LIN {X 0,Y 305.463,Z 118.06,A -85,B 0,C 180,E1 -16139.051,E2 -16139.051} C_VEL
LIN {X 0,Y 305.415,Z 118.064,A -85,B 0,C 180,E1 -16141.953,E2 -16141.953} C_VEL
LIN {X 0,Y 305.449,Z 118.063,A -85,B 0,C 180,E1 -16145.112,E2 -16145.112} C_VEL
LIN {X 0,Y 305.493,Z 118.055,A -85,B 0,C 180,E1 -16146.531,E2 -16146.531} C_VEL
LIN {X 0,Y 304.825,Z 118.142,A -85,B 0,C 180,E1 -16147.631,E2 -16147.631} C_VEL
LIN {X 0,Y 301.946,Z 118.499,A -85,B 0,C 180,E1 -16149.419,E2 -16149.419} C_VEL
LIN {X 0,Y 299.512,Z 118.803,A -85,B 0,C 180,E1 -16150.871,E2 -16150.871} C_VEL
LIN {X 0,Y 298.486,Z 118.925,A -85,B 0,C 180,E1 -16151.996,E2 -16151.996} C_VEL
LIN {X 0,Y 298.412,Z 118.928,A -85,B 0,C 180,E1 -16152.377,E2 -16152.377} C_VEL
LIN {X 0,Y 298.464,Z 118.93,A -85,B 0,C 180,E1 -16155.064,E2 -16155.064} C_VEL
LIN {X 0,Y 298.429,Z 118.934,A -85,B 0,C 180,E1 -16158.9,E2 -16158.9} C_VEL
LIN {X 0,Y 298.444,Z 118.927,A -85,B 0,C 180,E1 -16163.189,E2 -16163.189} C_VEL
LIN {X 0,Y 298.373,Z 118.94,A -85,B 0,C 180,E1 -16167.204,E2 -16167.204} C_VEL
LIN {X 0,Y 298.409,Z 118.927,A -85,B 0,C 180,E1 -16170.618,E2 -16170.618} C_VEL
LIN {X 0,Y 298.463,Z 118.924,A -85,B 0,C 180,E1 -16173.477,E2 -16173.477} C_VEL
LIN {X 0,Y 298.499,Z 118.926,A -85,B 0,C 180,E1 -16176.664,E2 -16176.664} C_VEL
LIN {X 0,Y 298.548,Z 118.918,A -85,B 0,C 180,E1 -16180.763,E2 -16180.763} C_VEL
LIN {X 0,Y 298.576,Z 118.913,A -85,B 0,C 180,E1 -16184.999,E2 -16184.999} C_VEL
LIN {X 0,Y 298.58,Z 118.916,A -85,B 0,C 180,E1 -16189.151,E2 -16189.151} C_VEL
LIN {X 0,Y 298.744,Z 118.888,A -85,B 0,C 180,E1 -16191.89,E2 -16191.89} C_VEL
LIN {X 0,Y 298.65,Z 118.896,A -85,B 0,C 180,E1 -16194.603,E2 -16194.603} C_VEL
LIN {X 0,Y 298.917,Z 118.873,A -85,B 0,C 180,E1 -16198.657,E2 -16198.657} C_VEL
LIN {X 0,Y 298.915,Z 118.874,A -85,B 0,C 180,E1 -16201.352,E2 -16201.352} C_VEL
LIN {X 0,Y 298.789,Z 118.885,A -85,B 0,C 180,E1 -16206.758,E2 -16206.758} C_VEL
LIN {X 0,Y 298.673,Z 118.905,A -85,B 0,C 180,E1 -16209.485,E2 -16209.485} C_VEL
LIN {X 0,Y 298.546,Z 118.92,A -85,B 0,C 180,E1 -16213.62,E2 -16213.62} C_VEL
LIN {X 0,Y 298.544,Z 118.921,A -85,B 0,C 180,E1 -16216.413,E2 -16216.413} C_VEL
LIN {X 0,Y 298.508,Z 118.924,A -85,B 0,C 180,E1 -16219.659,E2 -16219.659} C_VEL
LIN {X 0,Y 298.455,Z 118.93,A -85,B 0,C 180,E1 -16223.602,E2 -16223.602} C_VEL
LIN {X 0,Y 298.488,Z 118.928,A -85,B 0,C 180,E1 -16226.578,E2 -16226.578} C_VEL
LIN {X 0,Y 298.42,Z 118.934,A -85,B 0,C 180,E1 -16229.645,E2 -16229.645} C_VEL
LIN {X 0,Y 298.395,Z 118.938,A -85,B 0,C 180,E1 -16232.804,E2 -16232.804} C_VEL
LIN {X 0,Y 298.447,Z 118.932,A -85,B 0,C 180,E1 -16236.811,E2 -16236.811} C_VEL
LIN {X 0,Y 298.41,Z 118.936,A -85,B 0,C 180,E1 -16239.49,E2 -16239.49} C_VEL
LIN {X 0,Y 298.401,Z 118.939,A -85,B 0,C 180,E1 -16243.107,E2 -16243.107} C_VEL
LIN {X 0,Y 298.406,Z 118.938,A -85,B 0,C 180,E1 -16246.924,E2 -16246.924} C_VEL
LIN {X 0,Y 298.408,Z 118.938,A -85,B 0,C 180,E1 -16251.01,E2 -16251.01} C_VEL
LIN {X 0,Y 298.469,Z 119.026,A -85,B 0,C 180,E1 -16254.32,E2 -16254.32} C_VEL
LIN {X 0,Y 301.25,Z 131.247,A -85,B 0,C 180,E1 -16257.947,E2 -16257.947} C_VEL
LIN {X 0,Y 302.367,Z 136.348,A -85,B 0,C 180,E1 -16259.403,E2 -16259.403} C_VEL
LIN {X 0,Y 308.581,Z 152.762,A -85,B 0,C 180,E1 -16260.374,E2 -16260.374} C_VEL
LIN {X 0,Y 313.309,Z 184.218,A -85,B 0,C 180,E1 -16261.555,E2 -16261.555} C_VEL
LIN {X 0,Y 310.762,Z 275.009,A -85,B 0,C 180,E1 -16263.654,E2 -16263.654} C_VEL
LIN {X 0,Y 309.864,Z 288.738,A -85,B 0,C 180,E1 -16264.205,E2 -16264.205} C_VEL
LIN {X 0,Y 308.586,Z 302.3,A -85,B 0,C 180,E1 -16264.993,E2 -16264.993} C_VEL
LIN {X 0,Y 307.177,Z 315.166,A -85,B 0,C 180,E1 -16266.002,E2 -16266.002} C_VEL
LIN {X 0,Y 305.517,Z 328.379,A -85,B 0,C 180,E1 -16267.339,E2 -16267.339} C_VEL
LIN {X 0,Y 303.999,Z 338.844,A -85,B 0,C 180,E1 -16268.649,E2 -16268.649} C_VEL
LIN {X 0,Y 302.26,Z 349.716,A -85,B 0,C 180,E1 -16270.299,E2 -16270.299} C_VEL
LIN {X 0,Y 300.609,Z 360.479,A -85,B 0,C 180,E1 -16272.308,E2 -16272.308} C_VEL
LIN {X 0,Y 299.312,Z 369.247,A -85,B 0,C 180,E1 -16274.311,E2 -16274.311} C_VEL
LIN {X 0,Y 298.447,Z 375.565,A -85,B 0,C 180,E1 -16276.034,E2 -16276.034} C_VEL
LIN {X 0,Y 297.482,Z 382.796,A -85,B 0,C 180,E1 -16278.418,E2 -16278.418} C_VEL
LIN {X 0,Y 296.859,Z 389.274,A -85,B 0,C 180,E1 -16281.15,E2 -16281.15} C_VEL
LIN {X 0,Y 296.62,Z 392.996,A -85,B 0,C 180,E1 -16283.198,E2 -16283.198} C_VEL
LIN {X 0,Y 296.508,Z 396.618,A -85,B 0,C 180,E1 -16285.924,E2 -16285.924} C_VEL
LIN {X 0,Y 296.53,Z 397.888,A -85,B 0,C 180,E1 -16287.285,E2 -16287.285} C_VEL
LIN {X 0,Y 296.524,Z 399.388,A -85,B 0,C 180,E1 -16290.002,E2 -16290.002} C_VEL
LIN {X 0,Y 296.525,Z 399.54,A -85,B 0,C 180,E1 -16292.719,E2 -16292.719} C_VEL
LIN {X 0,Y 296.525,Z 398.363,A -85,B 0,C 180,E1 -16295.442,E2 -16295.442} C_VEL
LIN {X 0,Y 296.863,Z 395.854,A -85,B 0,C 180,E1 -16298.168,E2 -16298.168} C_VEL
LIN {X 0,Y 297.526,Z 391.948,A -85,B 0,C 180,E1 -16300.895,E2 -16300.895} C_VEL
LIN {X 0,Y 298.381,Z 387.999,A -85,B 0,C 180,E1 -16302.932,E2 -16302.932} C_VEL
LIN {X 0,Y 299.567,Z 383.169,A -85,B 0,C 180,E1 -16304.957,E2 -16304.957} C_VEL
LIN {X 0,Y 301.265,Z 376.222,A -85,B 0,C 180,E1 -16307.312,E2 -16307.312} C_VEL
LIN {X 0,Y 303.49,Z 367.688,A -85,B 0,C 180,E1 -16309.622,E2 -16309.622} C_VEL
LIN {X 0,Y 305.826,Z 358.785,A -85,B 0,C 180,E1 -16311.575,E2 -16311.575} C_VEL
LIN {X 0,Y 308.109,Z 349.971,A -85,B 0,C 180,E1 -16313.173,E2 -16313.173} C_VEL
LIN {X 0,Y 310.534,Z 339.507,A -85,B 0,C 180,E1 -16314.754,E2 -16314.754} C_VEL
LIN {X 0,Y 312.969,Z 328.052,A -85,B 0,C 180,E1 -16316.162,E2 -16316.162} C_VEL
LIN {X 0,Y 315.302,Z 315.733,A -85,B 0,C 180,E1 -16317.371,E2 -16317.371} C_VEL
LIN {X 0,Y 317.224,Z 303.024,A -85,B 0,C 180,E1 -16318.357,E2 -16318.357} C_VEL
LIN {X 0,Y 319.163,Z 288.698,A -85,B 0,C 180,E1 -16319.158,E2 -16319.158} C_VEL
LIN {X 0,Y 320.329,Z 275.633,A -85,B 0,C 180,E1 -16319.673,E2 -16319.673} C_VEL
LIN {X 0,Y 321.397,Z 250.364,A -85,B 0,C 180,E1 -16320.292,E2 -16320.292} C_VEL
LIN {X 0,Y 323.754,Z 186.86,A -85,B 0,C 180,E1 -16321.729,E2 -16321.729} C_VEL
LIN {X 0,Y 320.712,Z 169.862,A -85,B 0,C 180,E1 -16322.611,E2 -16322.611} C_VEL
LIN {X 0,Y 314.466,Z 156.405,A -85,B 0,C 180,E1 -16323.882,E2 -16323.882} C_VEL
LIN {X 0,Y 307.49,Z 143.185,A -85,B 0,C 180,E1 -16325.342,E2 -16325.342} C_VEL
LIN {X 0,Y 304.773,Z 138.364,A -85,B 0,C 180,E1 -16325.93,E2 -16325.93} C_VEL
LIN {X 0,Y 303.138,Z 135.112,A -85,B 0,C 180,E1 -16326.337,E2 -16326.337} C_VEL
LIN {X 0,Y 300.715,Z 126.551,A -85,B 0,C 180,E1 -16329.53,E2 -16329.53} C_VEL
LIN {X 0,Y 298.433,Z 118.935,A -85,B 0,C 180,E1 -16332.701,E2 -16332.701} C_VEL
LIN {X 0,Y 298.391,Z 118.937,A -85,B 0,C 180,E1 -16336.914,E2 -16336.914} C_VEL
LIN {X 0,Y 298.412,Z 118.938,A -85,B 0,C 180,E1 -16341.007,E2 -16341.007} C_VEL
LIN {X 0,Y 298.421,Z 118.938,A -85,B 0,C 180,E1 -16343.926,E2 -16343.926} C_VEL
LIN {X 0,Y 298.408,Z 118.94,A -85,B 0,C 180,E1 -16347.197,E2 -16347.197} C_VEL
LIN {X 0,Y 298.418,Z 118.938,A -85,B 0,C 180,E1 -16350.623,E2 -16350.623} C_VEL
LIN {X 0,Y 298.456,Z 118.93,A -85,B 0,C 180,E1 -16354.917,E2 -16354.917} C_VEL
LIN {X 0,Y 298.451,Z 118.924,A -85,B 0,C 180,E1 -16359.311,E2 -16359.311} C_VEL
LIN {X 0,Y 298.549,Z 118.922,A -85,B 0,C 180,E1 -16362.176,E2 -16362.176} C_VEL
LIN {X 0,Y 298.607,Z 118.908,A -85,B 0,C 180,E1 -16364.991,E2 -16364.991} C_VEL
LIN {X 0,Y 298.595,Z 118.909,A -85,B 0,C 180,E1 -16369.143,E2 -16369.143} C_VEL
LIN {X 0,Y 298.709,Z 118.893,A -85,B 0,C 180,E1 -16371.88,E2 -16371.88} C_VEL
LIN {X 0,Y 298.645,Z 118.911,A -85,B 0,C 180,E1 -16374.594,E2 -16374.594} C_VEL
LIN {X 0,Y 298.926,Z 118.876,A -85,B 0,C 180,E1 -16378.648,E2 -16378.648} C_VEL
LIN {X 0,Y 298.926,Z 118.862,A -85,B 0,C 180,E1 -16381.343,E2 -16381.343} C_VEL
LIN {X 0,Y 298.645,Z 118.899,A -85,B 0,C 180,E1 -16385.397,E2 -16385.397} C_VEL
LIN {X 0,Y 298.717,Z 118.898,A -85,B 0,C 180,E1 -16388.11,E2 -16388.11} C_VEL
LIN {X 0,Y 298.553,Z 118.917,A -85,B 0,C 180,E1 -16392.227,E2 -16392.227} C_VEL
LIN {X 0,Y 298.607,Z 118.916,A -85,B 0,C 180,E1 -16395.204,E2 -16395.204} C_VEL
LIN {X 0,Y 298.538,Z 118.92,A -85,B 0,C 180,E1 -16399.238,E2 -16399.238} C_VEL
LIN {X 0,Y 298.454,Z 118.929,A -85,B 0,C 180,E1 -16403.592,E2 -16403.592} C_VEL
LIN {X 0,Y 298.48,Z 118.925,A -85,B 0,C 180,E1 -16406.569,E2 -16406.569} C_VEL
LIN {X 0,Y 298.397,Z 118.919,A -85,B 0,C 180,E1 -16409.637,E2 -16409.637} C_VEL
LIN {X 0,Y 298.384,Z 118.937,A -85,B 0,C 180,E1 -16412.795,E2 -16412.795} C_VEL
LIN {X 0,Y 298.434,Z 119.032,A -85,B 0,C 180,E1 -16415.333,E2 -16415.333} C_VEL
LIN {X 0,Y 299.696,Z 123.328,A -85,B 0,C 180,E1 -16417.147,E2 -16417.147} C_VEL
LIN {X 0,Y 302.219,Z 127.458,A -85,B 0,C 180,E1 -16417.718,E2 -16417.718} C_VEL
LIN {X 0,Y 310.622,Z 141.607,A -85,B 0,C 180,E1 -16419.523,E2 -16419.523} C_VEL
LIN {X 0,Y 318.57,Z 156.631,A -85,B 0,C 180,E1 -16421.139,E2 -16421.139} C_VEL
LIN {X 0,Y 324.357,Z 169.063,A -85,B 0,C 180,E1 -16422.282,E2 -16422.282} C_VEL
LIN {X 0,Y 320.9,Z 259.44,A -85,B 0,C 180,E1 -16424.357,E2 -16424.357} C_VEL
LIN {X 0,Y 319.7,Z 273.914,A -85,B 0,C 180,E1 -16424.926,E2 -16424.926} C_VEL
LIN {X 0,Y 318.002,Z 288.36,A -85,B 0,C 180,E1 -16425.767,E2 -16425.767} C_VEL
LIN {X 0,Y 316.179,Z 301.192,A -85,B 0,C 180,E1 -16426.786,E2 -16426.786} C_VEL
LIN {X 0,Y 313.949,Z 313.553,A -85,B 0,C 180,E1 -16428.025,E2 -16428.025} C_VEL
LIN {X 0,Y 311.417,Z 325.585,A -85,B 0,C 180,E1 -16429.536,E2 -16429.536} C_VEL
LIN {X 0,Y 308.855,Z 336.611,A -85,B 0,C 180,E1 -16431.26,E2 -16431.26} C_VEL
LIN {X 0,Y 306.169,Z 347.321,A -85,B 0,C 180,E1 -16433.355,E2 -16433.355} C_VEL
LIN {X 0,Y 303.827,Z 356.079,A -85,B 0,C 180,E1 -16435.476,E2 -16435.476} C_VEL
LIN {X 0,Y 301.81,Z 363.266,A -85,B 0,C 180,E1 -16437.615,E2 -16437.615} C_VEL
LIN {X 0,Y 300.013,Z 369.838,A -85,B 0,C 180,E1 -16440.071,E2 -16440.071} C_VEL
LIN {X 0,Y 298.577,Z 375.202,A -85,B 0,C 180,E1 -16442.676,E2 -16442.676} C_VEL
LIN {X 0,Y 297.69,Z 378.573,A -85,B 0,C 180,E1 -16444.85,E2 -16444.85} C_VEL
LIN {X 0,Y 296.918,Z 381.627,A -85,B 0,C 180,E1 -16447.744,E2 -16447.744} C_VEL
LIN {X 0,Y 296.434,Z 383.173,A -85,B 0,C 180,E1 -16450.613,E2 -16450.613} C_VEL
LIN {X 0,Y 296.355,Z 383.402,A -85,B 0,C 180,E1 -16452.042,E2 -16452.042} C_VEL
LIN {X 0,Y 296.27,Z 382.793,A -85,B 0,C 180,E1 -16454.872,E2 -16454.872} C_VEL
LIN {X 0,Y 296.35,Z 381.8,A -85,B 0,C 180,E1 -16456.461,E2 -16456.461} C_VEL
LIN {X 0,Y 296.511,Z 379.191,A -85,B 0,C 180,E1 -16459.068,E2 -16459.068} C_VEL
LIN {X 0,Y 297.015,Z 374.96,A -85,B 0,C 180,E1 -16461.836,E2 -16461.836} C_VEL
LIN {X 0,Y 297.663,Z 369.164,A -85,B 0,C 180,E1 -16464.579,E2 -16464.579} C_VEL
LIN {X 0,Y 298.585,Z 362.628,A -85,B 0,C 180,E1 -16466.962,E2 -16466.962} C_VEL
LIN {X 0,Y 299.812,Z 354.531,A -85,B 0,C 180,E1 -16469.327,E2 -16469.327} C_VEL
LIN {X 0,Y 301.206,Z 346.043,A -85,B 0,C 180,E1 -16471.335,E2 -16471.335} C_VEL
LIN {X 0,Y 302.605,Z 337.211,A -85,B 0,C 180,E1 -16473.071,E2 -16473.071} C_VEL
LIN {X 0,Y 304.139,Z 326.644,A -85,B 0,C 180,E1 -16474.803,E2 -16474.803} C_VEL
LIN {X 0,Y 305.924,Z 314.369,A -85,B 0,C 180,E1 -16476.428,E2 -16476.428} C_VEL
LIN {X 0,Y 307.463,Z 302.214,A -85,B 0,C 180,E1 -16477.716,E2 -16477.716} C_VEL
LIN {X 0,Y 308.856,Z 288.771,A -85,B 0,C 180,E1 -16478.833,E2 -16478.833} C_VEL
LIN {X 0,Y 309.997,Z 274.732,A -85,B 0,C 180,E1 -16479.705,E2 -16479.705} C_VEL
LIN {X 0,Y 310.751,Z 261.089,A -85,B 0,C 180,E1 -16480.298,E2 -16480.298} C_VEL
LIN {X 0,Y 311.486,Z 239.443,A -85,B 0,C 180,E1 -16480.849,E2 -16480.849} C_VEL
LIN {X 0,Y 313.804,Z 159.13,A -85,B 0,C 180,E1 -16482.665,E2 -16482.665} C_VEL
LIN {X 0,Y 305.648,Z 137.375,A -85,B 0,C 180,E1 -16483.911,E2 -16483.911} C_VEL
LIN {X 0,Y 299.264,Z 122.065,A -85,B 0,C 180,E1 -16484.898,E2 -16484.898} C_VEL
LIN {X 0,Y 298.54,Z 118.93,A -85,B 0,C 180,E1 -16485.92,E2 -16485.92} C_VEL
LIN {X 0,Y 298.531,Z 118.927,A -85,B 0,C 180,E1 -16489.684,E2 -16489.684} C_VEL
LIN {X 0,Y 298.455,Z 118.935,A -85,B 0,C 180,E1 -16493.596,E2 -16493.596} C_VEL
LIN {X 0,Y 298.456,Z 118.931,A -85,B 0,C 180,E1 -16496.575,E2 -16496.575} C_VEL
LIN {X 0,Y 298.389,Z 118.941,A -85,B 0,C 180,E1 -16499.642,E2 -16499.642} C_VEL
LIN {X 0,Y 298.366,Z 118.944,A -85,B 0,C 180,E1 -16502.801,E2 -16502.801} C_VEL
LIN {X 0,Y 298.46,Z 118.933,A -85,B 0,C 180,E1 -16506.821,E2 -16506.821} C_VEL
LIN {X 0,Y 298.437,Z 118.934,A -85,B 0,C 180,E1 -16509.479,E2 -16509.479} C_VEL
LIN {X 0,Y 298.412,Z 118.928,A -85,B 0,C 180,E1 -16512.377,E2 -16512.377} C_VEL
LIN {X 0,Y 297.765,Z 119.011,A -85,B 0,C 180,E1 -16513.504,E2 -16513.504} C_VEL
LIN {X 0,Y 294.898,Z 119.372,A -85,B 0,C 180,E1 -16515.339,E2 -16515.339} C_VEL
LIN {X 0,Y 292.464,Z 119.68,A -85,B 0,C 180,E1 -16516.828,E2 -16516.828} C_VEL
LIN {X 0,Y 291.436,Z 119.805,A -85,B 0,C 180,E1 -16517.982,E2 -16517.982} C_VEL
LIN {X 0,Y 291.363,Z 119.816,A -85,B 0,C 180,E1 -16518.373,E2 -16518.373} C_VEL
LIN {X 0,Y 291.36,Z 119.804,A -85,B 0,C 180,E1 -16521.167,E2 -16521.167} C_VEL
LIN {X 0,Y 291.36,Z 119.816,A -85,B 0,C 180,E1 -16524.633,E2 -16524.633} C_VEL
LIN {X 0,Y 291.351,Z 119.816,A -85,B 0,C 180,E1 -16527.955,E2 -16527.955} C_VEL
LIN {X 0,Y 291.359,Z 119.801,A -85,B 0,C 180,E1 -16531.162,E2 -16531.162} C_VEL
LIN {X 0,Y 291.403,Z 119.809,A -85,B 0,C 180,E1 -16534.277,E2 -16534.277} C_VEL
LIN {X 0,Y 291.427,Z 119.807,A -85,B 0,C 180,E1 -16537.309,E2 -16537.309} C_VEL
LIN {X 0,Y 291.495,Z 119.799,A -85,B 0,C 180,E1 -16540.278,E2 -16540.278} C_VEL
LIN {X 0,Y 291.538,Z 119.79,A -85,B 0,C 180,E1 -16544.628,E2 -16544.628} C_VEL
LIN {X 0,Y 291.523,Z 119.794,A -85,B 0,C 180,E1 -16548.885,E2 -16548.885} C_VEL
LIN {X 0,Y 291.694,Z 119.767,A -85,B 0,C 180,E1 -16551.693,E2 -16551.693} C_VEL
LIN {X 0,Y 291.62,Z 119.77,A -85,B 0,C 180,E1 -16554.473,E2 -16554.473} C_VEL
LIN {X 0,Y 291.883,Z 119.749,A -85,B 0,C 180,E1 -16558.625,E2 -16558.625} C_VEL
LIN {X 0,Y 291.881,Z 119.749,A -85,B 0,C 180,E1 -16561.384,E2 -16561.384} C_VEL
LIN {X 0,Y 291.738,Z 119.763,A -85,B 0,C 180,E1 -16566.922,E2 -16566.922} C_VEL
LIN {X 0,Y 291.622,Z 119.782,A -85,B 0,C 180,E1 -16569.716,E2 -16569.716} C_VEL
LIN {X 0,Y 291.516,Z 119.795,A -85,B 0,C 180,E1 -16573.955,E2 -16573.955} C_VEL
LIN {X 0,Y 291.482,Z 119.801,A -85,B 0,C 180,E1 -16576.822,E2 -16576.822} C_VEL
LIN {X 0,Y 291.447,Z 119.804,A -85,B 0,C 180,E1 -16579.879,E2 -16579.879} C_VEL
LIN {X 0,Y 291.398,Z 119.811,A -85,B 0,C 180,E1 -16584.21,E2 -16584.21} C_VEL
LIN {X 0,Y 291.421,Z 119.803,A -85,B 0,C 180,E1 -16587.276,E2 -16587.276} C_VEL
LIN {X 0,Y 291.336,Z 119.82,A -85,B 0,C 180,E1 -16590.441,E2 -16590.441} C_VEL
LIN {X 0,Y 291.345,Z 119.816,A -85,B 0,C 180,E1 -16593.702,E2 -16593.702} C_VEL
LIN {X 0,Y 291.382,Z 119.812,A -85,B 0,C 180,E1 -16597.259,E2 -16597.259} C_VEL
LIN {X 0,Y 291.335,Z 119.815,A -85,B 0,C 180,E1 -16600.646,E2 -16600.646} C_VEL
LIN {X 0,Y 291.293,Z 119.826,A -85,B 0,C 180,E1 -16604.406,E2 -16604.406} C_VEL
LIN {X 0,Y 291.33,Z 119.816,A -85,B 0,C 180,E1 -16608.408,E2 -16608.408} C_VEL
LIN {X 0,Y 291.357,Z 119.817,A -85,B 0,C 180,E1 -16611.162,E2 -16611.162} C_VEL
LIN {X 0,Y 291.448,Z 119.827,A -85,B 0,C 180,E1 -16613.789,E2 -16613.789} C_VEL
LIN {X 0,Y 294.169,Z 131.986,A -85,B 0,C 180,E1 -16617.5,E2 -16617.5} C_VEL
LIN {X 0,Y 295.189,Z 136.326,A -85,B 0,C 180,E1 -16618.733,E2 -16618.733} C_VEL
LIN {X 0,Y 302.347,Z 155.276,A -85,B 0,C 180,E1 -16619.897,E2 -16619.897} C_VEL
LIN {X 0,Y 306.734,Z 184.058,A -85,B 0,C 180,E1 -16621.017,E2 -16621.017} C_VEL
LIN {X 0,Y 304.219,Z 273.974,A -85,B 0,C 180,E1 -16623.135,E2 -16623.135} C_VEL
LIN {X 0,Y 303.301,Z 287.998,A -85,B 0,C 180,E1 -16623.697,E2 -16623.697} C_VEL
LIN {X 0,Y 301.99,Z 301.707,A -85,B 0,C 180,E1 -16624.501,E2 -16624.501} C_VEL
LIN {X 0,Y 300.413,Z 315.56,A -85,B 0,C 180,E1 -16625.611,E2 -16625.611} C_VEL
LIN {X 0,Y 298.703,Z 328.667,A -85,B 0,C 180,E1 -16626.976,E2 -16626.976} C_VEL
LIN {X 0,Y 297.141,Z 339.053,A -85,B 0,C 180,E1 -16628.314,E2 -16628.314} C_VEL
LIN {X 0,Y 295.503,Z 348.87,A -85,B 0,C 180,E1 -16629.829,E2 -16629.829} C_VEL
LIN {X 0,Y 293.758,Z 359.745,A -85,B 0,C 180,E1 -16631.882,E2 -16631.882} C_VEL
LIN {X 0,Y 292.283,Z 369.374,A -85,B 0,C 180,E1 -16634.123,E2 -16634.123} C_VEL
LIN {X 0,Y 291.309,Z 376.142,A -85,B 0,C 180,E1 -16636.041,E2 -16636.041} C_VEL
LIN {X 0,Y 290.474,Z 382.31,A -85,B 0,C 180,E1 -16638.134,E2 -16638.134} C_VEL
LIN {X 0,Y 289.808,Z 388.851,A -85,B 0,C 180,E1 -16640.933,E2 -16640.933} C_VEL
LIN {X 0,Y 289.553,Z 392.631,A -85,B 0,C 180,E1 -16643.031,E2 -16643.031} C_VEL
LIN {X 0,Y 289.41,Z 396.306,A -85,B 0,C 180,E1 -16645.824,E2 -16645.824} C_VEL
LIN {X 0,Y 289.457,Z 397.603,A -85,B 0,C 180,E1 -16647.219,E2 -16647.219} C_VEL
LIN {X 0,Y 289.442,Z 399.155,A -85,B 0,C 180,E1 -16650.002,E2 -16650.002} C_VEL
LIN {X 0,Y 289.429,Z 399.356,A -85,B 0,C 180,E1 -16652.786,E2 -16652.786} C_VEL
LIN {X 0,Y 289.449,Z 398.229,A -85,B 0,C 180,E1 -16655.575,E2 -16655.575} C_VEL
LIN {X 0,Y 289.794,Z 395.774,A -85,B 0,C 180,E1 -16658.369,E2 -16658.369} C_VEL
LIN {X 0,Y 290.522,Z 391.935,A -85,B 0,C 180,E1 -16661.161,E2 -16661.161} C_VEL
LIN {X 0,Y 291.445,Z 388.04,A -85,B 0,C 180,E1 -16663.245,E2 -16663.245} C_VEL
LIN {X 0,Y 293.16,Z 381.467,A -85,B 0,C 180,E1 -16666.005,E2 -16666.005} C_VEL
LIN {X 0,Y 295.047,Z 374.192,A -85,B 0,C 180,E1 -16668.4,E2 -16668.4} C_VEL
LIN {X 0,Y 297.568,Z 365.215,A -85,B 0,C 180,E1 -16670.751,E2 -16670.751} C_VEL
LIN {X 0,Y 300.112,Z 355.84,A -85,B 0,C 180,E1 -16672.732,E2 -16672.732} C_VEL
LIN {X 0,Y 302.79,Z 345.5,A -85,B 0,C 180,E1 -16674.515,E2 -16674.515} C_VEL
LIN {X 0,Y 305.429,Z 334.274,A -85,B 0,C 180,E1 -16676.092,E2 -16676.092} C_VEL
LIN {X 0,Y 308.125,Z 321.608,A -85,B 0,C 180,E1 -16677.51,E2 -16677.51} C_VEL
LIN {X 0,Y 310.295,Z 309.477,A -85,B 0,C 180,E1 -16678.587,E2 -16678.587} C_VEL
LIN {X 0,Y 312.129,Z 297.413,A -85,B 0,C 180,E1 -16679.417,E2 -16679.417} C_VEL
LIN {X 0,Y 313.88,Z 282.469,A -85,B 0,C 180,E1 -16680.16,E2 -16680.16} C_VEL
LIN {X 0,Y 314.965,Z 268.57,A -85,B 0,C 180,E1 -16680.601,E2 -16680.601} C_VEL
LIN {X 0,Y 318.039,Z 188.05,A -85,B 0,C 180,E1 -16682.464,E2 -16682.464} C_VEL
LIN {X 0,Y 315.295,Z 172.701,A -85,B 0,C 180,E1 -16683.287,E2 -16683.287} C_VEL
LIN {X 0,Y 308.733,Z 158.563,A -85,B 0,C 180,E1 -16684.681,E2 -16684.681} C_VEL
LIN {X 0,Y 300.876,Z 143.736,A -85,B 0,C 180,E1 -16686.413,E2 -16686.413} C_VEL
LIN {X 0,Y 297.687,Z 138.447,A -85,B 0,C 180,E1 -16687.137,E2 -16687.137} C_VEL
LIN {X 0,Y 295.821,Z 134.869,A -85,B 0,C 180,E1 -16687.608,E2 -16687.608} C_VEL
LIN {X 0,Y 293.561,Z 127.111,A -85,B 0,C 180,E1 -16690.661,E2 -16690.661} C_VEL
LIN {X 0,Y 291.324,Z 119.821,A -85,B 0,C 180,E1 -16693.799,E2 -16693.799} C_VEL
LIN {X 0,Y 291.314,Z 119.807,A -85,B 0,C 180,E1 -16697.502,E2 -16697.502} C_VEL
LIN {X 0,Y 291.36,Z 119.817,A -85,B 0,C 180,E1 -16701.155,E2 -16701.155} C_VEL
LIN {X 0,Y 291.371,Z 119.816,A -85,B 0,C 180,E1 -16704.623,E2 -16704.623} C_VEL
LIN {X 0,Y 291.381,Z 119.812,A -85,B 0,C 180,E1 -16707.948,E2 -16707.948} C_VEL
LIN {X 0,Y 291.36,Z 119.815,A -85,B 0,C 180,E1 -16711.152,E2 -16711.152} C_VEL
LIN {X 0,Y 291.375,Z 119.815,A -85,B 0,C 180,E1 -16714.264,E2 -16714.264} C_VEL
LIN {X 0,Y 291.387,Z 119.811,A -85,B 0,C 180,E1 -16717.296,E2 -16717.296} C_VEL
LIN {X 0,Y 291.473,Z 119.792,A -85,B 0,C 180,E1 -16720.267,E2 -16720.267} C_VEL
LIN {X 0,Y 291.554,Z 119.783,A -85,B 0,C 180,E1 -16724.631,E2 -16724.631} C_VEL
LIN {X 0,Y 291.541,Z 119.785,A -85,B 0,C 180,E1 -16728.877,E2 -16728.877} C_VEL
LIN {X 0,Y 291.663,Z 119.772,A -85,B 0,C 180,E1 -16731.683,E2 -16731.683} C_VEL
LIN {X 0,Y 291.614,Z 119.786,A -85,B 0,C 180,E1 -16734.464,E2 -16734.464} C_VEL
LIN {X 0,Y 291.892,Z 119.751,A -85,B 0,C 180,E1 -16738.616,E2 -16738.616} C_VEL
LIN {X 0,Y 291.893,Z 119.738,A -85,B 0,C 180,E1 -16741.375,E2 -16741.375} C_VEL
LIN {X 0,Y 291.664,Z 119.774,A -85,B 0,C 180,E1 -16746.551,E2 -16746.551} C_VEL
LIN {X 0,Y 291.572,Z 119.781,A -85,B 0,C 180,E1 -16749.709,E2 -16749.709} C_VEL
LIN {X 0,Y 291.524,Z 119.79,A -85,B 0,C 180,E1 -16753.945,E2 -16753.945} C_VEL
LIN {X 0,Y 291.488,Z 119.793,A -85,B 0,C 180,E1 -16756.812,E2 -16756.812} C_VEL
LIN {X 0,Y 291.45,Z 119.798,A -85,B 0,C 180,E1 -16759.869,E2 -16759.869} C_VEL
LIN {X 0,Y 291.395,Z 119.812,A -85,B 0,C 180,E1 -16764.2,E2 -16764.2} C_VEL
LIN {X 0,Y 291.41,Z 119.812,A -85,B 0,C 180,E1 -16767.267,E2 -16767.267} C_VEL
LIN {X 0,Y 291.316,Z 119.802,A -85,B 0,C 180,E1 -16770.433,E2 -16770.433} C_VEL
LIN {X 0,Y 291.371,Z 119.987,A -85,B 0,C 180,E1 -16774.229,E2 -16774.229} C_VEL
LIN {X 0,Y 292.495,Z 123.617,A -85,B 0,C 180,E1 -16775.844,E2 -16775.844} C_VEL
LIN {X 0,Y 294.842,Z 127.48,A -85,B 0,C 180,E1 -16776.411,E2 -16776.411} C_VEL
LIN {X 0,Y 301.819,Z 138.719,A -85,B 0,C 180,E1 -16778.01,E2 -16778.01} C_VEL
LIN {X 0,Y 308.948,Z 151.389,A -85,B 0,C 180,E1 -16779.557,E2 -16779.557} C_VEL
LIN {X 0,Y 316.269,Z 166.096,A -85,B 0,C 180,E1 -16781.084,E2 -16781.084} C_VEL
LIN {X 0,Y 318.672,Z 171.401,A -85,B 0,C 180,E1 -16781.574,E2 -16781.574} C_VEL
LIN {X 0,Y 315.078,Z 259.814,A -85,B 0,C 180,E1 -16783.628,E2 -16783.628} C_VEL
LIN {X 0,Y 313.818,Z 274.5,A -85,B 0,C 180,E1 -16784.22,E2 -16784.22} C_VEL
LIN {X 0,Y 312.097,Z 288.475,A -85,B 0,C 180,E1 -16785.045,E2 -16785.045} C_VEL
LIN {X 0,Y 310.256,Z 300.988,A -85,B 0,C 180,E1 -16786.049,E2 -16786.049} C_VEL
LIN {X 0,Y 308.037,Z 312.92,A -85,B 0,C 180,E1 -16787.251,E2 -16787.251} C_VEL
LIN {X 0,Y 305.368,Z 325.134,A -85,B 0,C 180,E1 -16788.789,E2 -16788.789} C_VEL
LIN {X 0,Y 302.703,Z 336.224,A -85,B 0,C 180,E1 -16790.535,E2 -16790.535} C_VEL
LIN {X 0,Y 300.067,Z 346.259,A -85,B 0,C 180,E1 -16792.484,E2 -16792.484} C_VEL
LIN {X 0,Y 297.552,Z 355.242,A -85,B 0,C 180,E1 -16794.64,E2 -16794.64} C_VEL
LIN {X 0,Y 295.406,Z 362.623,A -85,B 0,C 180,E1 -16796.823,E2 -16796.823} C_VEL
LIN {X 0,Y 293.651,Z 368.666,A -85,B 0,C 180,E1 -16799.03,E2 -16799.03} C_VEL
LIN {X 0,Y 292.218,Z 373.509,A -85,B 0,C 180,E1 -16801.246,E2 -16801.246} C_VEL
LIN {X 0,Y 291.233,Z 376.946,A -85,B 0,C 180,E1 -16803.223,E2 -16803.223} C_VEL
LIN {X 0,Y 290.311,Z 380.195,A -85,B 0,C 180,E1 -16805.696,E2 -16805.696} C_VEL
LIN {X 0,Y 289.939,Z 381.596,A -85,B 0,C 180,E1 -16807.178,E2 -16807.178} C_VEL
LIN {X 0,Y 289.401,Z 383.276,A -85,B 0,C 180,E1 -16810.122,E2 -16810.122} C_VEL
LIN {X 0,Y 289.294,Z 383.57,A -85,B 0,C 180,E1 -16811.588,E2 -16811.588} C_VEL
LIN {X 0,Y 289.171,Z 383.095,A -85,B 0,C 180,E1 -16814.492,E2 -16814.492} C_VEL
LIN {X 0,Y 289.289,Z 381.216,A -85,B 0,C 180,E1 -16817.369,E2 -16817.369} C_VEL
LIN {X 0,Y 289.599,Z 377.895,A -85,B 0,C 180,E1 -16820.217,E2 -16820.217} C_VEL
LIN {X 0,Y 289.999,Z 374.4,A -85,B 0,C 180,E1 -16822.338,E2 -16822.338} C_VEL
LIN {X 0,Y 290.539,Z 370.008,A -85,B 0,C 180,E1 -16824.446,E2 -16824.446} C_VEL
LIN {X 0,Y 291.422,Z 363.633,A -85,B 0,C 180,E1 -16826.888,E2 -16826.888} C_VEL
LIN {X 0,Y 292.683,Z 355.705,A -85,B 0,C 180,E1 -16829.31,E2 -16829.31} C_VEL
LIN {X 0,Y 294.084,Z 347.414,A -85,B 0,C 180,E1 -16831.367,E2 -16831.367} C_VEL
LIN {X 0,Y 295.785,Z 337.062,A -85,B 0,C 180,E1 -16833.476,E2 -16833.476} C_VEL
LIN {X 0,Y 297.388,Z 326.376,A -85,B 0,C 180,E1 -16835.252,E2 -16835.252} C_VEL
LIN {X 0,Y 299.066,Z 315.332,A -85,B 0,C 180,E1 -16836.746,E2 -16836.746} C_VEL
LIN {X 0,Y 300.639,Z 303.382,A -85,B 0,C 180,E1 -16838.061,E2 -16838.061} C_VEL
LIN {X 0,Y 302.06,Z 290.237,A -85,B 0,C 180,E1 -16839.203,E2 -16839.203} C_VEL
LIN {X 0,Y 303.25,Z 276.628,A -85,B 0,C 180,E1 -16840.092,E2 -16840.092} C_VEL
LIN {X 0,Y 304.11,Z 262.667,A -85,B 0,C 180,E1 -16840.736,E2 -16840.736} C_VEL
LIN {X 0,Y 304.795,Z 243.568,A -85,B 0,C 180,E1 -16841.259,E2 -16841.259} C_VEL
LIN {X 0,Y 307.278,Z 160.711,A -85,B 0,C 180,E1 -16843.169,E2 -16843.169} C_VEL
LIN {X 0,Y 299.691,Z 140.407,A -85,B 0,C 180,E1 -16844.37,E2 -16844.37} C_VEL
LIN {X 0,Y 292.982,Z 124.529,A -85,B 0,C 180,E1 -16845.431,E2 -16845.431} C_VEL
LIN {X 0,Y 292.079,Z 122.181,A -85,B 0,C 180,E1 -16845.608,E2 -16845.608} C_VEL
LIN {X 0,Y 291.482,Z 119.807,A -85,B 0,C 180,E1 -16846.459,E2 -16846.459} C_VEL
LIN {X 0,Y 291.462,Z 119.806,A -85,B 0,C 180,E1 -16849.899,E2 -16849.899} C_VEL
LIN {X 0,Y 291.404,Z 119.81,A -85,B 0,C 180,E1 -16854.203,E2 -16854.203} C_VEL
LIN {X 0,Y 291.389,Z 119.811,A -85,B 0,C 180,E1 -16857.272,E2 -16857.272} C_VEL
LIN {X 0,Y 291.306,Z 119.821,A -85,B 0,C 180,E1 -16860.438,E2 -16860.438} C_VEL
LIN {X 0,Y 291.319,Z 119.821,A -85,B 0,C 180,E1 -16863.699,E2 -16863.699} C_VEL
LIN {X 0,Y 291.425,Z 119.809,A -85,B 0,C 180,E1 -16867.277,E2 -16867.277} C_VEL
LIN {X 0,Y 291.393,Z 119.813,A -85,B 0,C 180,E1 -16870.629,E2 -16870.629} C_VEL
LIN {X 0,Y 291.383,Z 119.804,A -85,B 0,C 180,E1 -16874.381,E2 -16874.381} C_VEL
LIN {X 0,Y 291.363,Z 119.816,A -85,B 0,C 180,E1 -16878.373,E2 -16878.373} C_VEL
LIN {X 0,Y 290.714,Z 119.901,A -85,B 0,C 180,E1 -16879.528,E2 -16879.528} C_VEL
LIN {X 0,Y 287.844,Z 120.252,A -85,B 0,C 180,E1 -16881.407,E2 -16881.407} C_VEL
LIN {X 0,Y 285.414,Z 120.55,A -85,B 0,C 180,E1 -16882.933,E2 -16882.933} C_VEL
LIN {X 0,Y 284.398,Z 120.678,A -85,B 0,C 180,E1 -16884.116,E2 -16884.116} C_VEL
LIN {X 0,Y 284.33,Z 120.689,A -85,B 0,C 180,E1 -16884.517,E2 -16884.517} C_VEL
LIN {X 0,Y 284.274,Z 120.693,A -85,B 0,C 180,E1 -16888.73,E2 -16888.73} C_VEL
LIN {X 0,Y 284.375,Z 120.678,A -85,B 0,C 180,E1 -16892.83,E2 -16892.83} C_VEL
LIN {X 0,Y 284.382,Z 120.685,A -85,B 0,C 180,E1 -16896.714,E2 -16896.714} C_VEL
LIN {X 0,Y 284.417,Z 120.68,A -85,B 0,C 180,E1 -16899.875,E2 -16899.875} C_VEL
LIN {X 0,Y 284.475,Z 120.67,A -85,B 0,C 180,E1 -16904.463,E2 -16904.463} C_VEL
LIN {X 0,Y 284.475,Z 120.672,A -85,B 0,C 180,E1 -16908.606,E2 -16908.606} C_VEL
LIN {X 0,Y 284.645,Z 120.646,A -85,B 0,C 180,E1 -16911.486,E2 -16911.486} C_VEL
LIN {X 0,Y 284.591,Z 120.645,A -85,B 0,C 180,E1 -16914.336,E2 -16914.336} C_VEL
LIN {X 0,Y 284.849,Z 120.625,A -85,B 0,C 180,E1 -16918.591,E2 -16918.591} C_VEL
LIN {X 0,Y 284.847,Z 120.624,A -85,B 0,C 180,E1 -16921.418,E2 -16921.418} C_VEL
LIN {X 0,Y 284.69,Z 120.642,A -85,B 0,C 180,E1 -16927.095,E2 -16927.095} C_VEL
LIN {X 0,Y 284.559,Z 120.662,A -85,B 0,C 180,E1 -16929.96,E2 -16929.96} C_VEL
LIN {X 0,Y 284.476,Z 120.673,A -85,B 0,C 180,E1 -16934.307,E2 -16934.307} C_VEL
LIN {X 0,Y 284.421,Z 120.679,A -85,B 0,C 180,E1 -16937.253,E2 -16937.253} C_VEL
LIN {X 0,Y 284.375,Z 120.686,A -85,B 0,C 180,E1 -16940.247,E2 -16940.247} C_VEL
LIN {X 0,Y 284.367,Z 120.685,A -85,B 0,C 180,E1 -16943.88,E2 -16943.88} C_VEL
LIN {X 0,Y 284.396,Z 120.678,A -85,B 0,C 180,E1 -16947.178,E2 -16947.178} C_VEL
LIN {X 0,Y 284.295,Z 120.692,A -85,B 0,C 180,E1 -16951.279,E2 -16951.279} C_VEL
LIN {X 0,Y 284.342,Z 120.688,A -85,B 0,C 180,E1 -16955.352,E2 -16955.352} C_VEL
LIN {X 0,Y 284.32,Z 120.695,A -85,B 0,C 180,E1 -16958.172,E2 -16958.172} C_VEL
LIN {X 0,Y 284.272,Z 120.7,A -85,B 0,C 180,E1 -16962.128,E2 -16962.128} C_VEL
LIN {X 0,Y 284.259,Z 120.703,A -85,B 0,C 180,E1 -16966.193,E2 -16966.193} C_VEL
LIN {X 0,Y 284.311,Z 120.698,A -85,B 0,C 180,E1 -16970.028,E2 -16970.028} C_VEL
LIN {X 0,Y 284.41,Z 120.848,A -85,B 0,C 180,E1 -16973.298,E2 -16973.298} C_VEL
LIN {X 0,Y 287.144,Z 132.928,A -85,B 0,C 180,E1 -16977.095,E2 -16977.095} C_VEL
LIN {X 0,Y 287.809,Z 135.936,A -85,B 0,C 180,E1 -16978.006,E2 -16978.006} C_VEL
LIN {X 0,Y 296.067,Z 157.207,A -85,B 0,C 180,E1 -16979.378,E2 -16979.378} C_VEL
LIN {X 0,Y 300.269,Z 185.672,A -85,B 0,C 180,E1 -16980.509,E2 -16980.509} C_VEL
LIN {X 0,Y 297.637,Z 274.127,A -85,B 0,C 180,E1 -16982.634,E2 -16982.634} C_VEL
LIN {X 0,Y 296.706,Z 288.028,A -85,B 0,C 180,E1 -16983.208,E2 -16983.208} C_VEL
LIN {X 0,Y 295.284,Z 302.247,A -85,B 0,C 180,E1 -16984.068,E2 -16984.068} C_VEL
LIN {X 0,Y 293.734,Z 315.075,A -85,B 0,C 180,E1 -16985.117,E2 -16985.117} C_VEL
LIN {X 0,Y 292.1,Z 327.49,A -85,B 0,C 180,E1 -16986.424,E2 -16986.424} C_VEL
LIN {X 0,Y 290.483,Z 338.05,A -85,B 0,C 180,E1 -16987.79,E2 -16987.79} C_VEL
LIN {X 0,Y 288.783,Z 348.005,A -85,B 0,C 180,E1 -16989.339,E2 -16989.339} C_VEL
LIN {X 0,Y 287.206,Z 357.333,A -85,B 0,C 180,E1 -16991.083,E2 -16991.083} C_VEL
LIN {X 0,Y 285.736,Z 366.614,A -85,B 0,C 180,E1 -16993.189,E2 -16993.189} C_VEL
LIN {X 0,Y 284.614,Z 374.435,A -85,B 0,C 180,E1 -16995.341,E2 -16995.341} C_VEL
LIN {X 0,Y 283.476,Z 381.806,A -85,B 0,C 180,E1 -16997.837,E2 -16997.837} C_VEL
LIN {X 0,Y 282.866,Z 386.962,A -85,B 0,C 180,E1 -16999.986,E2 -16999.986} C_VEL
LIN {X 0,Y 282.554,Z 391.076,A -85,B 0,C 180,E1 -17002.139,E2 -17002.139} C_VEL
LIN {X 0,Y 282.346,Z 394.811,A -85,B 0,C 180,E1 -17004.687,E2 -17004.687} C_VEL
LIN {X 0,Y 282.361,Z 397.314,A -85,B 0,C 180,E1 -17007.149,E2 -17007.149} C_VEL
LIN {X 0,Y 282.361,Z 398.919,A -85,B 0,C 180,E1 -17010.002,E2 -17010.002} C_VEL
LIN {X 0,Y 282.335,Z 399.173,A -85,B 0,C 180,E1 -17012.856,E2 -17012.856} C_VEL
LIN {X 0,Y 282.356,Z 398.099,A -85,B 0,C 180,E1 -17015.716,E2 -17015.716} C_VEL
LIN {X 0,Y 282.745,Z 395.699,A -85,B 0,C 180,E1 -17018.579,E2 -17018.579} C_VEL
LIN {X 0,Y 283.5,Z 391.916,A -85,B 0,C 180,E1 -17021.441,E2 -17021.441} C_VEL
LIN {X 0,Y 284.942,Z 386.645,A -85,B 0,C 180,E1 -17024.281,E2 -17024.281} C_VEL
LIN {X 0,Y 286.321,Z 381.572,A -85,B 0,C 180,E1 -17026.398,E2 -17026.398} C_VEL
LIN {X 0,Y 288.306,Z 374.37,A -85,B 0,C 180,E1 -17028.846,E2 -17028.846} C_VEL
LIN {X 0,Y 290.933,Z 365.511,A -85,B 0,C 180,E1 -17031.247,E2 -17031.247} C_VEL
LIN {X 0,Y 293.595,Z 356.257,A -85,B 0,C 180,E1 -17033.266,E2 -17033.266} C_VEL
LIN {X 0,Y 296.371,Z 346.056,A -85,B 0,C 180,E1 -17035.082,E2 -17035.082} C_VEL
LIN {X 0,Y 299.165,Z 334.729,A -85,B 0,C 180,E1 -17036.719,E2 -17036.719} C_VEL
LIN {X 0,Y 301.889,Z 322.525,A -85,B 0,C 180,E1 -17038.129,E2 -17038.129} C_VEL
LIN {X 0,Y 304.156,Z 310.672,A -85,B 0,C 180,E1 -17039.219,E2 -17039.219} C_VEL
LIN {X 0,Y 306.041,Z 299.032,A -85,B 0,C 180,E1 -17040.062,E2 -17040.062} C_VEL
LIN {X 0,Y 307.876,Z 284.808,A -85,B 0,C 180,E1 -17040.812,E2 -17040.812} C_VEL
LIN {X 0,Y 309.087,Z 271.045,A -85,B 0,C 180,E1 -17041.295,E2 -17041.295} C_VEL
LIN {X 0,Y 312.305,Z 188.821,A -85,B 0,C 180,E1 -17043.248,E2 -17043.248} C_VEL
LIN {X 0,Y 310.04,Z 175.819,A -85,B 0,C 180,E1 -17043.965,E2 -17043.965} C_VEL
LIN {X 0,Y 303.584,Z 161.806,A -85,B 0,C 180,E1 -17045.396,E2 -17045.396} C_VEL
LIN {X 0,Y 295.975,Z 147.484,A -85,B 0,C 180,E1 -17047.143,E2 -17047.143} C_VEL
LIN {X 0,Y 290.891,Z 138.828,A -85,B 0,C 180,E1 -17048.363,E2 -17048.363} C_VEL
LIN {X 0,Y 288.521,Z 134.506,A -85,B 0,C 180,E1 -17049.009,E2 -17049.009} C_VEL
LIN {X 0,Y 286.019,Z 126.209,A -85,B 0,C 180,E1 -17052.506,E2 -17052.506} C_VEL
LIN {X 0,Y 284.26,Z 120.699,A -85,B 0,C 180,E1 -17055.062,E2 -17055.062} C_VEL
LIN {X 0,Y 284.274,Z 120.677,A -85,B 0,C 180,E1 -17058.12,E2 -17058.12} C_VEL
LIN {X 0,Y 284.319,Z 120.692,A -85,B 0,C 180,E1 -17061.828,E2 -17061.828} C_VEL
LIN {X 0,Y 284.323,Z 120.687,A -85,B 0,C 180,E1 -17065.349,E2 -17065.349} C_VEL
LIN {X 0,Y 284.301,Z 120.689,A -85,B 0,C 180,E1 -17068.722,E2 -17068.722} C_VEL
LIN {X 0,Y 284.299,Z 120.688,A -85,B 0,C 180,E1 -17071.982,E2 -17071.982} C_VEL
LIN {X 0,Y 284.336,Z 120.681,A -85,B 0,C 180,E1 -17076.144,E2 -17076.144} C_VEL
LIN {X 0,Y 284.403,Z 120.672,A -85,B 0,C 180,E1 -17079.895,E2 -17079.895} C_VEL
LIN {X 0,Y 284.492,Z 120.662,A -85,B 0,C 180,E1 -17084.466,E2 -17084.466} C_VEL
LIN {X 0,Y 284.495,Z 120.661,A -85,B 0,C 180,E1 -17088.597,E2 -17088.597} C_VEL
LIN {X 0,Y 284.62,Z 120.651,A -85,B 0,C 180,E1 -17091.476,E2 -17091.476} C_VEL
LIN {X 0,Y 284.583,Z 120.661,A -85,B 0,C 180,E1 -17094.326,E2 -17094.326} C_VEL
LIN {X 0,Y 284.858,Z 120.627,A -85,B 0,C 180,E1 -17098.582,E2 -17098.582} C_VEL
LIN {X 0,Y 284.859,Z 120.614,A -85,B 0,C 180,E1 -17101.409,E2 -17101.409} C_VEL
LIN {X 0,Y 284.658,Z 120.651,A -85,B 0,C 180,E1 -17107.086,E2 -17107.086} C_VEL
LIN {X 0,Y 284.518,Z 120.661,A -85,B 0,C 180,E1 -17109.952,E2 -17109.952} C_VEL
LIN {X 0,Y 284.484,Z 120.67,A -85,B 0,C 180,E1 -17114.297,E2 -17114.297} C_VEL
LIN {X 0,Y 284.426,Z 120.673,A -85,B 0,C 180,E1 -17117.243,E2 -17117.243} C_VEL
LIN {X 0,Y 284.379,Z 120.679,A -85,B 0,C 180,E1 -17120.236,E2 -17120.236} C_VEL
LIN {X 0,Y 284.365,Z 120.684,A -85,B 0,C 180,E1 -17123.869,E2 -17123.869} C_VEL
LIN {X 0,Y 284.387,Z 120.686,A -85,B 0,C 180,E1 -17127.166,E2 -17127.166} C_VEL
LIN {X 0,Y 284.279,Z 120.687,A -85,B 0,C 180,E1 -17131.27,E2 -17131.27} C_VEL
LIN {X 0,Y 284.296,Z 120.708,A -85,B 0,C 180,E1 -17132.94,E2 -17132.94} C_VEL
LIN {X 0,Y 285.319,Z 124.019,A -85,B 0,C 180,E1 -17134.449,E2 -17134.449} C_VEL
LIN {X 0,Y 288.286,Z 128.494,A -85,B 0,C 180,E1 -17135.202,E2 -17135.202} C_VEL
LIN {X 0,Y 297.122,Z 142.761,A -85,B 0,C 180,E1 -17137.328,E2 -17137.328} C_VEL
LIN {X 0,Y 303.705,Z 154.543,A -85,B 0,C 180,E1 -17138.82,E2 -17138.82} C_VEL
LIN {X 0,Y 310.425,Z 168.001,A -85,B 0,C 180,E1 -17140.282,E2 -17140.282} C_VEL
LIN {X 0,Y 312.996,Z 173.708,A -85,B 0,C 180,E1 -17140.834,E2 -17140.834} C_VEL
LIN {X 0,Y 309.392,Z 259.081,A -85,B 0,C 180,E1 -17142.836,E2 -17142.836} C_VEL
LIN {X 0,Y 308.131,Z 273.792,A -85,B 0,C 180,E1 -17143.42,E2 -17143.42} C_VEL
LIN {X 0,Y 306.426,Z 287.393,A -85,B 0,C 180,E1 -17144.212,E2 -17144.212} C_VEL
LIN {X 0,Y 304.441,Z 300.367,A -85,B 0,C 180,E1 -17145.242,E2 -17145.242} C_VEL
LIN {X 0,Y 301.855,Z 313.819,A -85,B 0,C 180,E1 -17146.617,E2 -17146.617} C_VEL
LIN {X 0,Y 299.103,Z 325.912,A -85,B 0,C 180,E1 -17148.183,E2 -17148.183} C_VEL
LIN {X 0,Y 296.492,Z 336.218,A -85,B 0,C 180,E1 -17149.839,E2 -17149.839} C_VEL
LIN {X 0,Y 293.769,Z 346.189,A -85,B 0,C 180,E1 -17151.802,E2 -17151.802} C_VEL
LIN {X 0,Y 290.928,Z 355.724,A -85,B 0,C 180,E1 -17154.137,E2 -17154.137} C_VEL
LIN {X 0,Y 288.676,Z 363.046,A -85,B 0,C 180,E1 -17156.365,E2 -17156.365} C_VEL
LIN {X 0,Y 286.567,Z 369.901,A -85,B 0,C 180,E1 -17158.999,E2 -17158.999} C_VEL
LIN {X 0,Y 285.11,Z 374.567,A -85,B 0,C 180,E1 -17161.268,E2 -17161.268} C_VEL
LIN {X 0,Y 283.998,Z 378.191,A -85,B 0,C 180,E1 -17163.546,E2 -17163.546} C_VEL
LIN {X 0,Y 283.412,Z 380.089,A -85,B 0,C 180,E1 -17165.065,E2 -17165.065} C_VEL
LIN {X 0,Y 282.619,Z 382.658,A -85,B 0,C 180,E1 -17168.097,E2 -17168.097} C_VEL
LIN {X 0,Y 282.232,Z 383.74,A -85,B 0,C 180,E1 -17171.11,E2 -17171.11} C_VEL
LIN {X 0,Y 282.069,Z 383.394,A -85,B 0,C 180,E1 -17174.091,E2 -17174.091} C_VEL
LIN {X 0,Y 282.194,Z 381.639,A -85,B 0,C 180,E1 -17177.045,E2 -17177.045} C_VEL
LIN {X 0,Y 282.474,Z 378.473,A -85,B 0,C 180,E1 -17179.968,E2 -17179.968} C_VEL
LIN {X 0,Y 282.868,Z 375.088,A -85,B 0,C 180,E1 -17182.144,E2 -17182.144} C_VEL
LIN {X 0,Y 283.595,Z 369.212,A -85,B 0,C 180,E1 -17185.022,E2 -17185.022} C_VEL
LIN {X 0,Y 284.601,Z 362.59,A -85,B 0,C 180,E1 -17187.521,E2 -17187.521} C_VEL
LIN {X 0,Y 285.989,Z 354.366,A -85,B 0,C 180,E1 -17189.998,E2 -17189.998} C_VEL
LIN {X 0,Y 287.51,Z 345.759,A -85,B 0,C 180,E1 -17192.099,E2 -17192.099} C_VEL
LIN {X 0,Y 289.26,Z 335.344,A -85,B 0,C 180,E1 -17194.178,E2 -17194.178} C_VEL
LIN {X 0,Y 291.016,Z 323.736,A -85,B 0,C 180,E1 -17196.063,E2 -17196.063} C_VEL
LIN {X 0,Y 292.827,Z 312.075,A -85,B 0,C 180,E1 -17197.583,E2 -17197.583} C_VEL
LIN {X 0,Y 294.458,Z 299.304,A -85,B 0,C 180,E1 -17198.923,E2 -17198.923} C_VEL
LIN {X 0,Y 295.847,Z 286.079,A -85,B 0,C 180,E1 -17200.002,E2 -17200.002} C_VEL
LIN {X 0,Y 297.062,Z 271.655,A -85,B 0,C 180,E1 -17200.865,E2 -17200.865} C_VEL
LIN {X 0,Y 297.803,Z 257.197,A -85,B 0,C 180,E1 -17201.44,E2 -17201.44} C_VEL
LIN {X 0,Y 300.85,Z 162.691,A -85,B 0,C 180,E1 -17203.678,E2 -17203.678} C_VEL
LIN {X 0,Y 294.223,Z 144.524,A -85,B 0,C 180,E1 -17204.769,E2 -17204.769} C_VEL
LIN {X 0,Y 286.333,Z 125.789,A -85,B 0,C 180,E1 -17206.06,E2 -17206.06} C_VEL
LIN {X 0,Y 284.856,Z 122.469,A -85,B 0,C 180,E1 -17206.31,E2 -17206.31} C_VEL
LIN {X 0,Y 284.41,Z 120.689,A -85,B 0,C 180,E1 -17206.997,E2 -17206.997} C_VEL
LIN {X 0,Y 284.393,Z 120.685,A -85,B 0,C 180,E1 -17210.239,E2 -17210.239} C_VEL
LIN {X 0,Y 284.367,Z 120.688,A -85,B 0,C 180,E1 -17213.89,E2 -17213.89} C_VEL
LIN {X 0,Y 284.299,Z 120.694,A -85,B 0,C 180,E1 -17218.012,E2 -17218.012} C_VEL
LIN {X 0,Y 284.266,Z 120.703,A -85,B 0,C 180,E1 -17221.275,E2 -17221.275} C_VEL
LIN {X 0,Y 284.338,Z 120.691,A -85,B 0,C 180,E1 -17225.358,E2 -17225.358} C_VEL
LIN {X 0,Y 284.339,Z 120.689,A -85,B 0,C 180,E1 -17228.162,E2 -17228.162} C_VEL
LIN {X 0,Y 284.336,Z 120.688,A -85,B 0,C 180,E1 -17232.148,E2 -17232.148} C_VEL
LIN {X 0,Y 284.327,Z 120.689,A -85,B 0,C 180,E1 -17236.211,E2 -17236.211} C_VEL
LIN {X 0,Y 284.324,Z 120.688,A -85,B 0,C 180,E1 -17240.016,E2 -17240.016} C_VEL
LIN {X 0,Y 284.329,Z 120.684,A -85,B 0,C 180,E1 -17243.621,E2 -17243.621} C_VEL
LIN {X 0,Y 284.33,Z 120.689,A -85,B 0,C 180,E1 -17244.517,E2 -17244.517} C_VEL
LIN {X 0,Y 283.686,Z 120.778,A -85,B 0,C 180,E1 -17245.698,E2 -17245.698} C_VEL
LIN {X 0,Y 280.786,Z 121.135,A -85,B 0,C 180,E1 -17247.62,E2 -17247.62} C_VEL
LIN {X 0,Y 278.322,Z 121.433,A -85,B 0,C 180,E1 -17249.181,E2 -17249.181} C_VEL
LIN {X 0,Y 277.292,Z 121.555,A -85,B 0,C 180,E1 -17250.393,E2 -17250.393} C_VEL
LIN {X 0,Y 277.224,Z 121.559,A -85,B 0,C 180,E1 -17250.804,E2 -17250.804} C_VEL
LIN {X 0,Y 277.337,Z 121.553,A -85,B 0,C 180,E1 -17252.868,E2 -17252.868} C_VEL
LIN {X 0,Y 277.36,Z 121.562,A -85,B 0,C 180,E1 -17256.088,E2 -17256.088} C_VEL
LIN {X 0,Y 277.358,Z 121.557,A -85,B 0,C 180,E1 -17260.773,E2 -17260.773} C_VEL
LIN {X 0,Y 277.418,Z 121.549,A -85,B 0,C 180,E1 -17265.33,E2 -17265.33} C_VEL
LIN {X 0,Y 277.492,Z 121.542,A -85,B 0,C 180,E1 -17269.793,E2 -17269.793} C_VEL
LIN {X 0,Y 277.64,Z 121.512,A -85,B 0,C 180,E1 -17272.734,E2 -17272.734} C_VEL
LIN {X 0,Y 277.815,Z 121.501,A -85,B 0,C 180,E1 -17278.555,E2 -17278.555} C_VEL
LIN {X 0,Y 277.813,Z 121.5,A -85,B 0,C 180,E1 -17281.454,E2 -17281.454} C_VEL
LIN {X 0,Y 277.645,Z 121.521,A -85,B 0,C 180,E1 -17287.276,E2 -17287.276} C_VEL
LIN {X 0,Y 277.5,Z 121.541,A -85,B 0,C 180,E1 -17290.216,E2 -17290.216} C_VEL
LIN {X 0,Y 277.429,Z 121.553,A -85,B 0,C 180,E1 -17294.679,E2 -17294.679} C_VEL
LIN {X 0,Y 277.341,Z 121.563,A -85,B 0,C 180,E1 -17299.238,E2 -17299.238} C_VEL
LIN {X 0,Y 277.317,Z 121.565,A -85,B 0,C 180,E1 -17304.175,E2 -17304.175} C_VEL
LIN {X 0,Y 277.324,Z 121.558,A -85,B 0,C 180,E1 -17307.51,E2 -17307.51} C_VEL
LIN {X 0,Y 277.272,Z 121.571,A -85,B 0,C 180,E1 -17310.486,E2 -17310.486} C_VEL
LIN {X 0,Y 277.247,Z 121.573,A -85,B 0,C 180,E1 -17313.9,E2 -17313.9} C_VEL
LIN {X 0,Y 277.273,Z 121.57,A -85,B 0,C 180,E1 -17317.473,E2 -17317.473} C_VEL
LIN {X 0,Y 277.212,Z 121.573,A -85,B 0,C 180,E1 -17321.241,E2 -17321.241} C_VEL
LIN {X 0,Y 277.204,Z 121.58,A -85,B 0,C 180,E1 -17325.23,E2 -17325.23} C_VEL
LIN {X 0,Y 277.226,Z 121.575,A -85,B 0,C 180,E1 -17329.516,E2 -17329.516} C_VEL
LIN {X 0,Y 277.348,Z 121.731,A -85,B 0,C 180,E1 -17332.739,E2 -17332.739} C_VEL
LIN {X 0,Y 279.997,Z 133.256,A -85,B 0,C 180,E1 -17336.484,E2 -17336.484} C_VEL
LIN {X 0,Y 280.538,Z 135.754,A -85,B 0,C 180,E1 -17337.254,E2 -17337.254} C_VEL
LIN {X 0,Y 289.614,Z 158.671,A -85,B 0,C 180,E1 -17338.81,E2 -17338.81} C_VEL
LIN {X 0,Y 293.758,Z 185.628,A -85,B 0,C 180,E1 -17339.928,E2 -17339.928} C_VEL
LIN {X 0,Y 291.157,Z 273.003,A -85,B 0,C 180,E1 -17342.07,E2 -17342.07} C_VEL
LIN {X 0,Y 290.177,Z 287.28,A -85,B 0,C 180,E1 -17342.653,E2 -17342.653} C_VEL
LIN {X 0,Y 288.711,Z 301.641,A -85,B 0,C 180,E1 -17343.529,E2 -17343.529} C_VEL
LIN {X 0,Y 287.055,Z 314.914,A -85,B 0,C 180,E1 -17344.633,E2 -17344.633} C_VEL
LIN {X 0,Y 285.286,Z 328.052,A -85,B 0,C 180,E1 -17346.057,E2 -17346.057} C_VEL
LIN {X 0,Y 283.643,Z 338.237,A -85,B 0,C 180,E1 -17347.417,E2 -17347.417} C_VEL
LIN {X 0,Y 281.72,Z 349.118,A -85,B 0,C 180,E1 -17349.179,E2 -17349.179} C_VEL
LIN {X 0,Y 279.853,Z 359.887,A -85,B 0,C 180,E1 -17351.328,E2 -17351.328} C_VEL
LIN {X 0,Y 278.309,Z 369.382,A -85,B 0,C 180,E1 -17353.667,E2 -17353.667} C_VEL
LIN {X 0,Y 277.24,Z 376.118,A -85,B 0,C 180,E1 -17355.693,E2 -17355.693} C_VEL
LIN {X 0,Y 276.189,Z 383.136,A -85,B 0,C 180,E1 -17358.256,E2 -17358.256} C_VEL
LIN {X 0,Y 275.683,Z 387.975,A -85,B 0,C 180,E1 -17360.464,E2 -17360.464} C_VEL
LIN {X 0,Y 275.397,Z 391.88,A -85,B 0,C 180,E1 -17362.671,E2 -17362.671} C_VEL
LIN {X 0,Y 275.228,Z 395.671,A -85,B 0,C 180,E1 -17365.609,E2 -17365.609} C_VEL
LIN {X 0,Y 275.268,Z 397.023,A -85,B 0,C 180,E1 -17367.075,E2 -17367.075} C_VEL
LIN {X 0,Y 275.283,Z 398.683,A -85,B 0,C 180,E1 -17370.002,E2 -17370.002} C_VEL
LIN {X 0,Y 275.244,Z 398.99,A -85,B 0,C 180,E1 -17372.929,E2 -17372.929} C_VEL
LIN {X 0,Y 275.291,Z 397.97,A -85,B 0,C 180,E1 -17375.863,E2 -17375.863} C_VEL
LIN {X 0,Y 275.69,Z 395.623,A -85,B 0,C 180,E1 -17378.8,E2 -17378.8} C_VEL
LIN {X 0,Y 276.491,Z 391.897,A -85,B 0,C 180,E1 -17381.735,E2 -17381.735} C_VEL
LIN {X 0,Y 278.046,Z 386.699,A -85,B 0,C 180,E1 -17384.643,E2 -17384.643} C_VEL
LIN {X 0,Y 279.698,Z 380.977,A -85,B 0,C 180,E1 -17387.095,E2 -17387.095} C_VEL
LIN {X 0,Y 281.933,Z 373.455,A -85,B 0,C 180,E1 -17389.667,E2 -17389.667} C_VEL
LIN {X 0,Y 284.748,Z 364.382,A -85,B 0,C 180,E1 -17392.112,E2 -17392.112} C_VEL
LIN {X 0,Y 287.608,Z 354.93,A -85,B 0,C 180,E1 -17394.163,E2 -17394.163} C_VEL
LIN {X 0,Y 290.557,Z 344.556,A -85,B 0,C 180,E1 -17395.993,E2 -17395.993} C_VEL
LIN {X 0,Y 293.325,Z 333.516,A -85,B 0,C 180,E1 -17397.586,E2 -17397.586} C_VEL
LIN {X 0,Y 296.058,Z 321.871,A -85,B 0,C 180,E1 -17398.928,E2 -17398.928} C_VEL
LIN {X 0,Y 298.351,Z 309.914,A -85,B 0,C 180,E1 -17400.04,E2 -17400.04} C_VEL
LIN {X 0,Y 300.54,Z 296.815,A -85,B 0,C 180,E1 -17400.963,E2 -17400.963} C_VEL
LIN {X 0,Y 302.432,Z 281.802,A -85,B 0,C 180,E1 -17401.722,E2 -17401.722} C_VEL
LIN {X 0,Y 303.555,Z 267.782,A -85,B 0,C 180,E1 -17402.177,E2 -17402.177} C_VEL
LIN {X 0,Y 306.781,Z 190.338,A -85,B 0,C 180,E1 -17404.023,E2 -17404.023} C_VEL
LIN {X 0,Y 304.85,Z 179.001,A -85,B 0,C 180,E1 -17404.665,E2 -17404.665} C_VEL
LIN {X 0,Y 298.837,Z 165.884,A -85,B 0,C 180,E1 -17406.05,E2 -17406.05} C_VEL
LIN {X 0,Y 291.921,Z 152.605,A -85,B 0,C 180,E1 -17407.704,E2 -17407.704} C_VEL
LIN {X 0,Y 285.69,Z 141.949,A -85,B 0,C 180,E1 -17409.261,E2 -17409.261} C_VEL
LIN {X 0,Y 283.138,Z 137.821,A -85,B 0,C 180,E1 -17409.925,E2 -17409.925} C_VEL
LIN {X 0,Y 281.133,Z 134.181,A -85,B 0,C 180,E1 -17410.542,E2 -17410.542} C_VEL
LIN {X 0,Y 278.708,Z 126.359,A -85,B 0,C 180,E1 -17414.051,E2 -17414.051} C_VEL
LIN {X 0,Y 277.233,Z 121.58,A -85,B 0,C 180,E1 -17416.447,E2 -17416.447} C_VEL
LIN {X 0,Y 277.248,Z 121.567,A -85,B 0,C 180,E1 -17420.67,E2 -17420.67} C_VEL
LIN {X 0,Y 277.294,Z 121.57,A -85,B 0,C 180,E1 -17424.338,E2 -17424.338} C_VEL
LIN {X 0,Y 277.256,Z 121.572,A -85,B 0,C 180,E1 -17427.834,E2 -17427.834} C_VEL
LIN {X 0,Y 277.255,Z 121.571,A -85,B 0,C 180,E1 -17431.204,E2 -17431.204} C_VEL
LIN {X 0,Y 277.262,Z 121.574,A -85,B 0,C 180,E1 -17434.47,E2 -17434.47} C_VEL
LIN {X 0,Y 277.281,Z 121.572,A -85,B 0,C 180,E1 -17437.65,E2 -17437.65} C_VEL
LIN {X 0,Y 277.357,Z 121.553,A -85,B 0,C 180,E1 -17440.763,E2 -17440.763} C_VEL
LIN {X 0,Y 277.442,Z 121.547,A -85,B 0,C 180,E1 -17445.322,E2 -17445.322} C_VEL
LIN {X 0,Y 277.47,Z 121.546,A -85,B 0,C 180,E1 -17449.783,E2 -17449.783} C_VEL
LIN {X 0,Y 277.612,Z 121.518,A -85,B 0,C 180,E1 -17452.723,E2 -17452.723} C_VEL
LIN {X 0,Y 277.825,Z 121.502,A -85,B 0,C 180,E1 -17458.546,E2 -17458.546} C_VEL
LIN {X 0,Y 277.825,Z 121.49,A -85,B 0,C 180,E1 -17461.445,E2 -17461.445} C_VEL
LIN {X 0,Y 277.616,Z 121.529,A -85,B 0,C 180,E1 -17467.267,E2 -17467.267} C_VEL
LIN {X 0,Y 277.461,Z 121.541,A -85,B 0,C 180,E1 -17470.208,E2 -17470.208} C_VEL
LIN {X 0,Y 277.437,Z 121.551,A -85,B 0,C 180,E1 -17474.669,E2 -17474.669} C_VEL
LIN {X 0,Y 277.345,Z 121.559,A -85,B 0,C 180,E1 -17479.228,E2 -17479.228} C_VEL
LIN {X 0,Y 277.324,Z 121.561,A -85,B 0,C 180,E1 -17483.915,E2 -17483.915} C_VEL
LIN {X 0,Y 277.315,Z 121.568,A -85,B 0,C 180,E1 -17487.497,E2 -17487.497} C_VEL
LIN {X 0,Y 277.238,Z 121.596,A -85,B 0,C 180,E1 -17491.622,E2 -17491.622} C_VEL
LIN {X 0,Y 278.062,Z 124.132,A -85,B 0,C 180,E1 -17492.898,E2 -17492.898} C_VEL
LIN {X 0,Y 280.42,Z 127.995,A -85,B 0,C 180,E1 -17493.562,E2 -17493.562} C_VEL
LIN {X 0,Y 282.03,Z 130.222,A -85,B 0,C 180,E1 -17493.988,E2 -17493.988} C_VEL
LIN {X 0,Y 288.291,Z 139.928,A -85,B 0,C 180,E1 -17495.601,E2 -17495.601} C_VEL
LIN {X 0,Y 295.593,Z 152.272,A -85,B 0,C 180,E1 -17497.37,E2 -17497.37} C_VEL
LIN {X 0,Y 303.42,Z 167.307,A -85,B 0,C 180,E1 -17499.17,E2 -17499.17} C_VEL
LIN {X 0,Y 307.395,Z 175.915,A -85,B 0,C 180,E1 -17500.058,E2 -17500.058} C_VEL
LIN {X 0,Y 303.682,Z 259.722,A -85,B 0,C 180,E1 -17502.057,E2 -17502.057} C_VEL
LIN {X 0,Y 302.386,Z 274.09,A -85,B 0,C 180,E1 -17502.639,E2 -17502.639} C_VEL
LIN {X 0,Y 300.636,Z 287.545,A -85,B 0,C 180,E1 -17503.434,E2 -17503.434} C_VEL
LIN {X 0,Y 298.403,Z 301.445,A -85,B 0,C 180,E1 -17504.563,E2 -17504.563} C_VEL
LIN {X 0,Y 295.917,Z 313.858,A -85,B 0,C 180,E1 -17505.86,E2 -17505.86} C_VEL
LIN {X 0,Y 293.17,Z 325.439,A -85,B 0,C 180,E1 -17507.371,E2 -17507.371} C_VEL
LIN {X 0,Y 290.237,Z 336.535,A -85,B 0,C 180,E1 -17509.169,E2 -17509.169} C_VEL
LIN {X 0,Y 287.314,Z 346.785,A -85,B 0,C 180,E1 -17511.237,E2 -17511.237} C_VEL
LIN {X 0,Y 284.335,Z 356.22,A -85,B 0,C 180,E1 -17513.612,E2 -17513.612} C_VEL
LIN {X 0,Y 281.965,Z 363.486,A -85,B 0,C 180,E1 -17515.886,E2 -17515.886} C_VEL
LIN {X 0,Y 279.664,Z 370.522,A -85,B 0,C 180,E1 -17518.684,E2 -17518.684} C_VEL
LIN {X 0,Y 278.005,Z 375.561,A -85,B 0,C 180,E1 -17521.291,E2 -17521.291} C_VEL
LIN {X 0,Y 277.214,Z 377.953,A -85,B 0,C 180,E1 -17522.847,E2 -17522.847} C_VEL
LIN {X 0,Y 276.066,Z 381.503,A -85,B 0,C 180,E1 -17525.961,E2 -17525.961} C_VEL
LIN {X 0,Y 275.67,Z 382.688,A -85,B 0,C 180,E1 -17527.515,E2 -17527.515} C_VEL
LIN {X 0,Y 275.178,Z 383.91,A -85,B 0,C 180,E1 -17530.607,E2 -17530.607} C_VEL
LIN {X 0,Y 274.983,Z 383.692,A -85,B 0,C 180,E1 -17533.67,E2 -17533.67} C_VEL
LIN {X 0,Y 275.081,Z 382.064,A -85,B 0,C 180,E1 -17536.704,E2 -17536.704} C_VEL
LIN {X 0,Y 275.319,Z 379.029,A -85,B 0,C 180,E1 -17539.705,E2 -17539.705} C_VEL
LIN {X 0,Y 275.735,Z 375.776,A -85,B 0,C 180,E1 -17541.939,E2 -17541.939} C_VEL
LIN {X 0,Y 276.262,Z 371.665,A -85,B 0,C 180,E1 -17544.158,E2 -17544.158} C_VEL
LIN {X 0,Y 276.993,Z 366.534,A -85,B 0,C 180,E1 -17546.361,E2 -17546.361} C_VEL
LIN {X 0,Y 278.208,Z 359.213,A -85,B 0,C 180,E1 -17548.912,E2 -17548.912} C_VEL
LIN {X 0,Y 279.833,Z 350.134,A -85,B 0,C 180,E1 -17551.437,E2 -17551.437} C_VEL
LIN {X 0,Y 281.511,Z 340.738,A -85,B 0,C 180,E1 -17553.552,E2 -17553.552} C_VEL
LIN {X 0,Y 283.267,Z 330.102,A -85,B 0,C 180,E1 -17555.515,E2 -17555.515} C_VEL
LIN {X 0,Y 285.173,Z 318.462,A -85,B 0,C 180,E1 -17557.254,E2 -17557.254} C_VEL
LIN {X 0,Y 287.027,Z 305.552,A -85,B 0,C 180,E1 -17558.801,E2 -17558.801} C_VEL
LIN {X 0,Y 288.718,Z 291.913,A -85,B 0,C 180,E1 -17560.074,E2 -17560.074} C_VEL
LIN {X 0,Y 289.935,Z 278.827,A -85,B 0,C 180,E1 -17561.003,E2 -17561.003} C_VEL
LIN {X 0,Y 290.911,Z 264.683,A -85,B 0,C 180,E1 -17561.715,E2 -17561.715} C_VEL
LIN {X 0,Y 291.604,Z 248.201,A -85,B 0,C 180,E1 -17562.216,E2 -17562.216} C_VEL
LIN {X 0,Y 294.296,Z 163.728,A -85,B 0,C 180,E1 -17564.244,E2 -17564.244} C_VEL
LIN {X 0,Y 286.775,Z 143.904,A -85,B 0,C 180,E1 -17565.508,E2 -17565.508} C_VEL
LIN {X 0,Y 280.589,Z 129.217,A -85,B 0,C 180,E1 -17566.563,E2 -17566.563} C_VEL
LIN {X 0,Y 277.583,Z 122.58,A -85,B 0,C 180,E1 -17567.114,E2 -17567.114} C_VEL
LIN {X 0,Y 277.362,Z 121.566,A -85,B 0,C 180,E1 -17567.509,E2 -17567.509} C_VEL
LIN {X 0,Y 277.321,Z 121.566,A -85,B 0,C 180,E1 -17570.779,E2 -17570.779} C_VEL
LIN {X 0,Y 277.331,Z 121.563,A -85,B 0,C 180,E1 -17574.192,E2 -17574.192} C_VEL
LIN {X 0,Y 277.293,Z 121.566,A -85,B 0,C 180,E1 -17577.506,E2 -17577.506} C_VEL
LIN {X 0,Y 277.24,Z 121.574,A -85,B 0,C 180,E1 -17580.483,E2 -17580.483} C_VEL
LIN {X 0,Y 277.225,Z 121.576,A -85,B 0,C 180,E1 -17583.896,E2 -17583.896} C_VEL
LIN {X 0,Y 277.292,Z 121.568,A -85,B 0,C 180,E1 -17587.463,E2 -17587.463} C_VEL
LIN {X 0,Y 277.276,Z 121.569,A -85,B 0,C 180,E1 -17591.221,E2 -17591.221} C_VEL
LIN {X 0,Y 277.263,Z 121.569,A -85,B 0,C 180,E1 -17595.21,E2 -17595.21} C_VEL
LIN {X 0,Y 277.268,Z 121.566,A -85,B 0,C 180,E1 -17599.498,E2 -17599.498} C_VEL
LIN {X 0,Y 277.264,Z 121.559,A -85,B 0,C 180,E1 -17602.538,E2 -17602.538} C_VEL
LIN {X 0,Y 277.23,Z 121.576,A -85,B 0,C 180,E1 -17606.109,E2 -17606.109} C_VEL
LIN {X 0,Y 277.238,Z 121.568,A -85,B 0,C 180,E1 -17609.542,E2 -17609.542} C_VEL
LIN {X 0,Y 277.224,Z 121.559,A -85,B 0,C 180,E1 -17610.804,E2 -17610.804} C_VEL
LIN {X 0,Y 276.612,Z 121.638,A -85,B 0,C 180,E1 -17612.016,E2 -17612.016} C_VEL
LIN {X 0,Y 273.82,Z 121.997,A -85,B 0,C 180,E1 -17613.993,E2 -17613.993} C_VEL
LIN {X 0,Y 271.407,Z 122.303,A -85,B 0,C 180,E1 -17615.598,E2 -17615.598} C_VEL
LIN {X 0,Y 270.344,Z 122.434,A -85,B 0,C 180,E1 -17616.842,E2 -17616.842} C_VEL
LIN {X 0,Y 270.244,Z 122.444,A -85,B 0,C 180,E1 -17617.264,E2 -17617.264} C_VEL
LIN {X 0,Y 270.313,Z 122.437,A -85,B 0,C 180,E1 -17620.251,E2 -17620.251} C_VEL
LIN {X 0,Y 270.386,Z 122.424,A -85,B 0,C 180,E1 -17624.94,E2 -17624.94} C_VEL
LIN {X 0,Y 270.427,Z 122.424,A -85,B 0,C 180,E1 -17629.524,E2 -17629.524} C_VEL
LIN {X 0,Y 270.598,Z 122.388,A -85,B 0,C 180,E1 -17632.544,E2 -17632.544} C_VEL
LIN {X 0,Y 270.78,Z 122.377,A -85,B 0,C 180,E1 -17638.518,E2 -17638.518} C_VEL
LIN {X 0,Y 270.779,Z 122.375,A -85,B 0,C 180,E1 -17641.492,E2 -17641.492} C_VEL
LIN {X 0,Y 270.603,Z 122.4,A -85,B 0,C 180,E1 -17647.466,E2 -17647.466} C_VEL
LIN {X 0,Y 270.435,Z 122.422,A -85,B 0,C 180,E1 -17650.486,E2 -17650.486} C_VEL
LIN {X 0,Y 270.398,Z 122.429,A -85,B 0,C 180,E1 -17655.069,E2 -17655.069} C_VEL
LIN {X 0,Y 270.298,Z 122.439,A -85,B 0,C 180,E1 -17659.76,E2 -17659.76} C_VEL
LIN {X 0,Y 270.272,Z 122.444,A -85,B 0,C 180,E1 -17664.59,E2 -17664.59} C_VEL
LIN {X 0,Y 270.271,Z 122.437,A -85,B 0,C 180,E1 -17667.913,E2 -17667.913} C_VEL
LIN {X 0,Y 270.184,Z 122.45,A -85,B 0,C 180,E1 -17671.353,E2 -17671.353} C_VEL
LIN {X 0,Y 270.203,Z 122.449,A -85,B 0,C 180,E1 -17674.91,E2 -17674.91} C_VEL
LIN {X 0,Y 270.2,Z 122.45,A -85,B 0,C 180,E1 -17678.715,E2 -17678.715} C_VEL
LIN {X 0,Y 270.168,Z 122.457,A -85,B 0,C 180,E1 -17683.253,E2 -17683.253} C_VEL
LIN {X 0,Y 270.176,Z 122.457,A -85,B 0,C 180,E1 -17687.446,E2 -17687.446} C_VEL
LIN {X 0,Y 270.256,Z 122.466,A -85,B 0,C 180,E1 -17692.097,E2 -17692.097} C_VEL
LIN {X 0,Y 272.67,Z 132.773,A -85,B 0,C 180,E1 -17695.573,E2 -17695.573} C_VEL
LIN {X 0,Y 273.338,Z 135.752,A -85,B 0,C 180,E1 -17696.471,E2 -17696.471} C_VEL
LIN {X 0,Y 281.963,Z 157.06,A -85,B 0,C 180,E1 -17698.01,E2 -17698.01} C_VEL
LIN {X 0,Y 283.836,Z 162.685,A -85,B 0,C 180,E1 -17698.357,E2 -17698.357} C_VEL
LIN {X 0,Y 287.334,Z 187.613,A -85,B 0,C 180,E1 -17699.39,E2 -17699.39} C_VEL
LIN {X 0,Y 284.535,Z 274.204,A -85,B 0,C 180,E1 -17701.562,E2 -17701.562} C_VEL
LIN {X 0,Y 283.488,Z 288.728,A -85,B 0,C 180,E1 -17702.203,E2 -17702.203} C_VEL
LIN {X 0,Y 281.924,Z 303.244,A -85,B 0,C 180,E1 -17703.141,E2 -17703.141} C_VEL
LIN {X 0,Y 280.341,Z 315.236,A -85,B 0,C 180,E1 -17704.18,E2 -17704.18} C_VEL
LIN {X 0,Y 278.632,Z 327.596,A -85,B 0,C 180,E1 -17705.552,E2 -17705.552} C_VEL
LIN {X 0,Y 276.986,Z 337.199,A -85,B 0,C 180,E1 -17706.843,E2 -17706.843} C_VEL
LIN {X 0,Y 275.212,Z 347.243,A -85,B 0,C 180,E1 -17708.466,E2 -17708.466} C_VEL
LIN {X 0,Y 273.363,Z 357.466,A -85,B 0,C 180,E1 -17710.477,E2 -17710.477} C_VEL
LIN {X 0,Y 271.767,Z 366.719,A -85,B 0,C 180,E1 -17712.701,E2 -17712.701} C_VEL
LIN {X 0,Y 270.569,Z 374.411,A -85,B 0,C 180,E1 -17714.947,E2 -17714.947} C_VEL
LIN {X 0,Y 269.517,Z 380.795,A -85,B 0,C 180,E1 -17717.196,E2 -17717.196} C_VEL
LIN {X 0,Y 268.796,Z 386.026,A -85,B 0,C 180,E1 -17719.456,E2 -17719.456} C_VEL
LIN {X 0,Y 268.42,Z 390.26,A -85,B 0,C 180,E1 -17721.722,E2 -17721.722} C_VEL
LIN {X 0,Y 268.167,Z 394.627,A -85,B 0,C 180,E1 -17724.833,E2 -17724.833} C_VEL
LIN {X 0,Y 268.178,Z 396.732,A -85,B 0,C 180,E1 -17726.998,E2 -17726.998} C_VEL
LIN {X 0,Y 268.207,Z 398.447,A -85,B 0,C 180,E1 -17730.002,E2 -17730.002} C_VEL
LIN {X 0,Y 268.155,Z 398.806,A -85,B 0,C 180,E1 -17733.007,E2 -17733.007} C_VEL
LIN {X 0,Y 268.223,Z 397.841,A -85,B 0,C 180,E1 -17736.018,E2 -17736.018} C_VEL
LIN {X 0,Y 268.652,Z 395.552,A -85,B 0,C 180,E1 -17739.033,E2 -17739.033} C_VEL
LIN {X 0,Y 269.495,Z 391.89,A -85,B 0,C 180,E1 -17742.044,E2 -17742.044} C_VEL
LIN {X 0,Y 271.142,Z 386.756,A -85,B 0,C 180,E1 -17745.025,E2 -17745.025} C_VEL
LIN {X 0,Y 273.077,Z 380.526,A -85,B 0,C 180,E1 -17747.769,E2 -17747.769} C_VEL
LIN {X 0,Y 275.244,Z 373.656,A -85,B 0,C 180,E1 -17750.166,E2 -17750.166} C_VEL
LIN {X 0,Y 278.193,Z 364.71,A -85,B 0,C 180,E1 -17752.662,E2 -17752.662} C_VEL
LIN {X 0,Y 281.166,Z 355.363,A -85,B 0,C 180,E1 -17754.753,E2 -17754.753} C_VEL
LIN {X 0,Y 284.509,Z 344.169,A -85,B 0,C 180,E1 -17756.766,E2 -17756.766} C_VEL
LIN {X 0,Y 287.425,Z 332.988,A -85,B 0,C 180,E1 -17758.399,E2 -17758.399} C_VEL
LIN {X 0,Y 290.258,Z 321.267,A -85,B 0,C 180,E1 -17759.762,E2 -17759.762} C_VEL
LIN {X 0,Y 292.622,Z 309.227,A -85,B 0,C 180,E1 -17760.891,E2 -17760.891} C_VEL
LIN {X 0,Y 294.941,Z 295.976,A -85,B 0,C 180,E1 -17761.819,E2 -17761.819} C_VEL
LIN {X 0,Y 296.79,Z 281.608,A -85,B 0,C 180,E1 -17762.548,E2 -17762.548} C_VEL
LIN {X 0,Y 297.924,Z 267.734,A -85,B 0,C 180,E1 -17763.007,E2 -17763.007} C_VEL
LIN {X 0,Y 301.216,Z 191.192,A -85,B 0,C 180,E1 -17764.864,E2 -17764.864} C_VEL
LIN {X 0,Y 299.562,Z 181.774,A -85,B 0,C 180,E1 -17765.426,E2 -17765.426} C_VEL
LIN {X 0,Y 293.558,Z 168.693,A -85,B 0,C 180,E1 -17766.872,E2 -17766.872} C_VEL
LIN {X 0,Y 286.064,Z 154.328,A -85,B 0,C 180,E1 -17768.753,E2 -17768.753} C_VEL
LIN {X 0,Y 279.431,Z 143.169,A -85,B 0,C 180,E1 -17770.509,E2 -17770.509} C_VEL
LIN {X 0,Y 276.471,Z 138.512,A -85,B 0,C 180,E1 -17771.331,E2 -17771.331} C_VEL
LIN {X 0,Y 273.837,Z 134.018,A -85,B 0,C 180,E1 -17772.12,E2 -17772.12} C_VEL
LIN {X 0,Y 271.474,Z 126.658,A -85,B 0,C 180,E1 -17775.65,E2 -17775.65} C_VEL
LIN {X 0,Y 270.155,Z 122.437,A -85,B 0,C 180,E1 -17777.852,E2 -17777.852} C_VEL
LIN {X 0,Y 270.225,Z 122.452,A -85,B 0,C 180,E1 -17781.372,E2 -17781.372} C_VEL
LIN {X 0,Y 270.214,Z 122.445,A -85,B 0,C 180,E1 -17785.092,E2 -17785.092} C_VEL
LIN {X 0,Y 270.201,Z 122.444,A -85,B 0,C 180,E1 -17789.134,E2 -17789.134} C_VEL
LIN {X 0,Y 270.239,Z 122.438,A -85,B 0,C 180,E1 -17792.16,E2 -17792.16} C_VEL
LIN {X 0,Y 270.243,Z 122.437,A -85,B 0,C 180,E1 -17795.54,E2 -17795.54} C_VEL
LIN {X 0,Y 270.315,Z 122.427,A -85,B 0,C 180,E1 -17800.241,E2 -17800.241} C_VEL
LIN {X 0,Y 270.41,Z 122.418,A -85,B 0,C 180,E1 -17804.931,E2 -17804.931} C_VEL
LIN {X 0,Y 270.422,Z 122.421,A -85,B 0,C 180,E1 -17809.514,E2 -17809.514} C_VEL
LIN {X 0,Y 270.574,Z 122.394,A -85,B 0,C 180,E1 -17812.533,E2 -17812.533} C_VEL
LIN {X 0,Y 270.789,Z 122.378,A -85,B 0,C 180,E1 -17818.508,E2 -17818.508} C_VEL
LIN {X 0,Y 270.791,Z 122.366,A -85,B 0,C 180,E1 -17821.482,E2 -17821.482} C_VEL
LIN {X 0,Y 270.576,Z 122.407,A -85,B 0,C 180,E1 -17827.457,E2 -17827.457} C_VEL
LIN {X 0,Y 270.414,Z 122.421,A -85,B 0,C 180,E1 -17830.477,E2 -17830.477} C_VEL
LIN {X 0,Y 270.405,Z 122.428,A -85,B 0,C 180,E1 -17835.059,E2 -17835.059} C_VEL
LIN {X 0,Y 270.302,Z 122.433,A -85,B 0,C 180,E1 -17839.75,E2 -17839.75} C_VEL
LIN {X 0,Y 270.27,Z 122.445,A -85,B 0,C 180,E1 -17844.58,E2 -17844.58} C_VEL
LIN {X 0,Y 270.263,Z 122.441,A -85,B 0,C 180,E1 -17847.903,E2 -17847.903} C_VEL
LIN {X 0,Y 270.232,Z 122.562,A -85,B 0,C 180,E1 -17850.231,E2 -17850.231} C_VEL
LIN {X 0,Y 270.803,Z 124.57,A -85,B 0,C 180,E1 -17851.225,E2 -17851.225} C_VEL
LIN {X 0,Y 273.627,Z 128.784,A -85,B 0,C 180,E1 -17852.066,E2 -17852.066} C_VEL
LIN {X 0,Y 274.86,Z 130.43,A -85,B 0,C 180,E1 -17852.416,E2 -17852.416} C_VEL
LIN {X 0,Y 277.464,Z 134.162,A -85,B 0,C 180,E1 -17853.147,E2 -17853.147} C_VEL
LIN {X 0,Y 285.886,Z 147.484,A -85,B 0,C 180,E1 -17855.395,E2 -17855.395} C_VEL
LIN {X 0,Y 293.928,Z 161.804,A -85,B 0,C 180,E1 -17857.388,E2 -17857.388} C_VEL
LIN {X 0,Y 301.029,Z 176.473,A -85,B 0,C 180,E1 -17859.069,E2 -17859.069} C_VEL
LIN {X 0,Y 301.868,Z 178.309,A -85,B 0,C 180,E1 -17859.262,E2 -17859.262} C_VEL
LIN {X 0,Y 298.043,Z 260.323,A -85,B 0,C 180,E1 -17861.245,E2 -17861.245} C_VEL
LIN {X 0,Y 296.629,Z 275.07,A -85,B 0,C 180,E1 -17861.861,E2 -17861.861} C_VEL
LIN {X 0,Y 294.731,Z 288.952,A -85,B 0,C 180,E1 -17862.712,E2 -17862.712} C_VEL
LIN {X 0,Y 292.408,Z 302.591,A -85,B 0,C 180,E1 -17863.857,E2 -17863.857} C_VEL
LIN {X 0,Y 289.64,Z 315.675,A -85,B 0,C 180,E1 -17865.275,E2 -17865.275} C_VEL
LIN {X 0,Y 286.508,Z 328.029,A -85,B 0,C 180,E1 -17866.978,E2 -17866.978} C_VEL
LIN {X 0,Y 283.349,Z 339.134,A -85,B 0,C 180,E1 -17868.904,E2 -17868.904} C_VEL
LIN {X 0,Y 280.144,Z 349.517,A -85,B 0,C 180,E1 -17871.155,E2 -17871.155} C_VEL
LIN {X 0,Y 277.339,Z 358.021,A -85,B 0,C 180,E1 -17873.449,E2 -17873.449} C_VEL
LIN {X 0,Y 274.548,Z 366.054,A -85,B 0,C 180,E1 -17876.165,E2 -17876.165} C_VEL
LIN {X 0,Y 272.364,Z 372.351,A -85,B 0,C 180,E1 -17878.928,E2 -17878.928} C_VEL
LIN {X 0,Y 270.515,Z 377.61,A -85,B 0,C 180,E1 -17882.031,E2 -17882.031} C_VEL
LIN {X 0,Y 269.712,Z 379.768,A -85,B 0,C 180,E1 -17883.704,E2 -17883.704} C_VEL
LIN {X 0,Y 268.706,Z 382.669,A -85,B 0,C 180,E1 -17886.899,E2 -17886.899} C_VEL
LIN {X 0,Y 268.128,Z 384.067,A -85,B 0,C 180,E1 -17890.075,E2 -17890.075} C_VEL
LIN {X 0,Y 267.886,Z 383.991,A -85,B 0,C 180,E1 -17893.225,E2 -17893.225} C_VEL
LIN {X 0,Y 267.954,Z 382.489,A -85,B 0,C 180,E1 -17896.344,E2 -17896.344} C_VEL
LIN {X 0,Y 268.173,Z 379.582,A -85,B 0,C 180,E1 -17899.427,E2 -17899.427} C_VEL
LIN {X 0,Y 268.765,Z 375.199,A -85,B 0,C 180,E1 -17902.485,E2 -17902.485} C_VEL
LIN {X 0,Y 269.329,Z 370.871,A -85,B 0,C 180,E1 -17904.758,E2 -17904.758} C_VEL
LIN {X 0,Y 270.307,Z 364.561,A -85,B 0,C 180,E1 -17907.39,E2 -17907.39} C_VEL
LIN {X 0,Y 271.703,Z 356.702,A -85,B 0,C 180,E1 -17909.998,E2 -17909.998} C_VEL
LIN {X 0,Y 273.279,Z 348.486,A -85,B 0,C 180,E1 -17912.209,E2 -17912.209} C_VEL
LIN {X 0,Y 275.055,Z 338.61,A -85,B 0,C 180,E1 -17914.394,E2 -17914.394} C_VEL
LIN {X 0,Y 276.886,Z 327.66,A -85,B 0,C 180,E1 -17916.374,E2 -17916.374} C_VEL
LIN {X 0,Y 278.971,Z 315.429,A -85,B 0,C 180,E1 -17918.145,E2 -17918.145} C_VEL
LIN {X 0,Y 280.722,Z 303.34,A -85,B 0,C 180,E1 -17919.545,E2 -17919.545} C_VEL
LIN {X 0,Y 282.287,Z 290,A -85,B 0,C 180,E1 -17920.76,E2 -17920.76} C_VEL
LIN {X 0,Y 283.622,Z 276.092,A -85,B 0,C 180,E1 -17921.703,E2 -17921.703} C_VEL
LIN {X 0,Y 284.571,Z 261.59,A -85,B 0,C 180,E1 -17922.387,E2 -17922.387} C_VEL
LIN {X 0,Y 285.456,Z 237.692,A -85,B 0,C 180,E1 -17923.037,E2 -17923.037} C_VEL
LIN {X 0,Y 287.918,Z 165.663,A -85,B 0,C 180,E1 -17924.792,E2 -17924.792} C_VEL
LIN {X 0,Y 281.843,Z 149.28,A -85,B 0,C 180,E1 -17925.857,E2 -17925.857} C_VEL
LIN {X 0,Y 274.989,Z 132.843,A -85,B 0,C 180,E1 -17927.067,E2 -17927.067} C_VEL
LIN {X 0,Y 270.497,Z 123.403,A -85,B 0,C 180,E1 -17927.855,E2 -17927.855} C_VEL
LIN {X 0,Y 270.325,Z 122.638,A -85,B 0,C 180,E1 -17927.976,E2 -17927.976} C_VEL
LIN {X 0,Y 270.241,Z 122.45,A -85,B 0,C 180,E1 -17931.349,E2 -17931.349} C_VEL
LIN {X 0,Y 270.259,Z 122.444,A -85,B 0,C 180,E1 -17934.585,E2 -17934.585} C_VEL
LIN {X 0,Y 270.24,Z 122.445,A -85,B 0,C 180,E1 -17937.91,E2 -17937.91} C_VEL
LIN {X 0,Y 270.153,Z 122.46,A -85,B 0,C 180,E1 -17941.349,E2 -17941.349} C_VEL
LIN {X 0,Y 270.191,Z 122.455,A -85,B 0,C 180,E1 -17944.904,E2 -17944.904} C_VEL
LIN {X 0,Y 270.248,Z 122.446,A -85,B 0,C 180,E1 -17948.734,E2 -17948.734} C_VEL
LIN {X 0,Y 270.24,Z 122.441,A -85,B 0,C 180,E1 -17952.542,E2 -17952.542} C_VEL
LIN {X 0,Y 270.206,Z 122.451,A -85,B 0,C 180,E1 -17956.738,E2 -17956.738} C_VEL
LIN {X 0,Y 270.222,Z 122.443,A -85,B 0,C 180,E1 -17959.451,E2 -17959.451} C_VEL
LIN {X 0,Y 270.232,Z 122.439,A -85,B 0,C 180,E1 -17963.725,E2 -17963.725} C_VEL
LIN {X 0,Y 270.18,Z 122.453,A -85,B 0,C 180,E1 -17966.897,E2 -17966.897} C_VEL
LIN {X 0,Y 270.17,Z 122.437,A -85,B 0,C 180,E1 -17970.806,E2 -17970.806} C_VEL
LIN {X 0,Y 270.248,Z 122.437,A -85,B 0,C 180,E1 -17973.769,E2 -17973.769} C_VEL
LIN {X 0,Y 270.244,Z 122.444,A -85,B 0,C 180,E1 -17977.264,E2 -17977.264} C_VEL
LIN {X 0,Y 269.56,Z 122.53,A -85,B 0,C 180,E1 -17978.508,E2 -17978.508} C_VEL
LIN {X 0,Y 266.773,Z 122.88,A -85,B 0,C 180,E1 -17980.538,E2 -17980.538} C_VEL
LIN {X 0,Y 264.425,Z 123.177,A -85,B 0,C 180,E1 -17982.188,E2 -17982.188} C_VEL
LIN {X 0,Y 263.415,Z 123.299,A -85,B 0,C 180,E1 -17983.464,E2 -17983.464} C_VEL
LIN {X 0,Y 263.33,Z 123.307,A -85,B 0,C 180,E1 -17983.897,E2 -17983.897} C_VEL
LIN {X 0,Y 263.322,Z 123.31,A -85,B 0,C 180,E1 -17987.677,E2 -17987.677} C_VEL
LIN {X 0,Y 263.544,Z 123.275,A -85,B 0,C 180,E1 -17990.798,E2 -17990.798} C_VEL
LIN {X 0,Y 263.503,Z 123.266,A -85,B 0,C 180,E1 -17993.881,E2 -17993.881} C_VEL
LIN {X 0,Y 263.744,Z 123.254,A -85,B 0,C 180,E1 -17998.478,E2 -17998.478} C_VEL
LIN {X 0,Y 263.743,Z 123.251,A -85,B 0,C 180,E1 -18001.532,E2 -18001.532} C_VEL
LIN {X 0,Y 263.565,Z 123.276,A -85,B 0,C 180,E1 -18007.667,E2 -18007.667} C_VEL
LIN {X 0,Y 263.368,Z 123.304,A -85,B 0,C 180,E1 -18010.771,E2 -18010.771} C_VEL
LIN {X 0,Y 263.346,Z 123.305,A -85,B 0,C 180,E1 -18015.483,E2 -18015.483} C_VEL
LIN {X 0,Y 263.26,Z 123.317,A -85,B 0,C 180,E1 -18020.311,E2 -18020.311} C_VEL
LIN {X 0,Y 263.207,Z 123.321,A -85,B 0,C 180,E1 -18025.296,E2 -18025.296} C_VEL
LIN {X 0,Y 263.179,Z 123.324,A -85,B 0,C 180,E1 -18028.734,E2 -18028.734} C_VEL
LIN {X 0,Y 263.133,Z 123.328,A -85,B 0,C 180,E1 -18032.293,E2 -18032.293} C_VEL
LIN {X 0,Y 263.186,Z 123.325,A -85,B 0,C 180,E1 -18036.768,E2 -18036.768} C_VEL
LIN {X 0,Y 263.127,Z 123.329,A -85,B 0,C 180,E1 -18041.598,E2 -18041.598} C_VEL
LIN {X 0,Y 263.109,Z 123.337,A -85,B 0,C 180,E1 -18046.159,E2 -18046.159} C_VEL
LIN {X 0,Y 263.111,Z 123.338,A -85,B 0,C 180,E1 -18050.132,E2 -18050.132} C_VEL
LIN {X 0,Y 263.204,Z 123.479,A -85,B 0,C 180,E1 -18051.518,E2 -18051.518} C_VEL
LIN {X 0,Y 265.519,Z 133.085,A -85,B 0,C 180,E1 -18054.873,E2 -18054.873} C_VEL
LIN {X 0,Y 266.098,Z 135.571,A -85,B 0,C 180,E1 -18055.631,E2 -18055.631} C_VEL
LIN {X 0,Y 274.538,Z 156.083,A -85,B 0,C 180,E1 -18057.203,E2 -18057.203} C_VEL
LIN {X 0,Y 277.661,Z 164.828,A -85,B 0,C 180,E1 -18057.789,E2 -18057.789} C_VEL
LIN {X 0,Y 280.907,Z 188.525,A -85,B 0,C 180,E1 -18058.795,E2 -18058.795} C_VEL
LIN {X 0,Y 278.039,Z 274.155,A -85,B 0,C 180,E1 -18060.99,E2 -18060.99} C_VEL
LIN {X 0,Y 277.023,Z 287.86,A -85,B 0,C 180,E1 -18061.599,E2 -18061.599} C_VEL
LIN {X 0,Y 275.545,Z 301.407,A -85,B 0,C 180,E1 -18062.467,E2 -18062.467} C_VEL
LIN {X 0,Y 273.64,Z 315.542,A -85,B 0,C 180,E1 -18063.705,E2 -18063.705} C_VEL
LIN {X 0,Y 271.829,Z 328.084,A -85,B 0,C 180,E1 -18065.142,E2 -18065.142} C_VEL
LIN {X 0,Y 269.998,Z 338.535,A -85,B 0,C 180,E1 -18066.615,E2 -18066.615} C_VEL
LIN {X 0,Y 267.958,Z 349.305,A -85,B 0,C 180,E1 -18068.46,E2 -18068.46} C_VEL
LIN {X 0,Y 265.982,Z 359.986,A -85,B 0,C 180,E1 -18070.716,E2 -18070.716} C_VEL
LIN {X 0,Y 264.308,Z 369.468,A -85,B 0,C 180,E1 -18073.196,E2 -18073.196} C_VEL
LIN {X 0,Y 263.012,Z 377.184,A -85,B 0,C 180,E1 -18075.692,E2 -18075.692} C_VEL
LIN {X 0,Y 261.943,Z 383.899,A -85,B 0,C 180,E1 -18078.394,E2 -18078.394} C_VEL
LIN {X 0,Y 261.366,Z 389.843,A -85,B 0,C 180,E1 -18081.497,E2 -18081.497} C_VEL
LIN {X 0,Y 261.145,Z 393.258,A -85,B 0,C 180,E1 -18083.822,E2 -18083.822} C_VEL
LIN {X 0,Y 261.091,Z 396.437,A -85,B 0,C 180,E1 -18086.916,E2 -18086.916} C_VEL
LIN {X 0,Y 261.123,Z 397.495,A -85,B 0,C 180,E1 -18088.46,E2 -18088.46} C_VEL
LIN {X 0,Y 261.133,Z 398.209,A -85,B 0,C 180,E1 -18090.002,E2 -18090.002} C_VEL
LIN {X 0,Y 261.112,Z 398.584,A -85,B 0,C 180,E1 -18091.545,E2 -18091.545} C_VEL
LIN {X 0,Y 261.032,Z 398.333,A -85,B 0,C 180,E1 -18094.635,E2 -18094.635} C_VEL
LIN {X 0,Y 261.306,Z 396.767,A -85,B 0,C 180,E1 -18097.731,E2 -18097.731} C_VEL
LIN {X 0,Y 261.997,Z 393.86,A -85,B 0,C 180,E1 -18100.825,E2 -18100.825} C_VEL
LIN {X 0,Y 263.307,Z 389.539,A -85,B 0,C 180,E1 -18103.902,E2 -18103.902} C_VEL
LIN {X 0,Y 265.284,Z 383.685,A -85,B 0,C 180,E1 -18106.945,E2 -18106.945} C_VEL
LIN {X 0,Y 267.439,Z 377.135,A -85,B 0,C 180,E1 -18109.578,E2 -18109.578} C_VEL
LIN {X 0,Y 270.271,Z 369.056,A -85,B 0,C 180,E1 -18112.153,E2 -18112.153} C_VEL
LIN {X 0,Y 273.146,Z 360.632,A -85,B 0,C 180,E1 -18114.312,E2 -18114.312} C_VEL
LIN {X 0,Y 276.513,Z 350.496,A -85,B 0,C 180,E1 -18116.412,E2 -18116.412} C_VEL
LIN {X 0,Y 279.791,Z 339.29,A -85,B 0,C 180,E1 -18118.288,E2 -18118.288} C_VEL
LIN {X 0,Y 282.705,Z 328.015,A -85,B 0,C 180,E1 -18119.817,E2 -18119.817} C_VEL
LIN {X 0,Y 285.568,Z 315.825,A -85,B 0,C 180,E1 -18121.121,E2 -18121.121} C_VEL
LIN {X 0,Y 287.995,Z 303.421,A -85,B 0,C 180,E1 -18122.163,E2 -18122.163} C_VEL
LIN {X 0,Y 290.253,Z 289.606,A -85,B 0,C 180,E1 -18123.013,E2 -18123.013} C_VEL
LIN {X 0,Y 291.862,Z 275.257,A -85,B 0,C 180,E1 -18123.633,E2 -18123.633} C_VEL
LIN {X 0,Y 292.949,Z 255.346,A -85,B 0,C 180,E1 -18124.175,E2 -18124.175} C_VEL
LIN {X 0,Y 295.813,Z 192.741,A -85,B 0,C 180,E1 -18125.699,E2 -18125.699} C_VEL
LIN {X 0,Y 294.406,Z 184.809,A -85,B 0,C 180,E1 -18126.195,E2 -18126.195} C_VEL
LIN {X 0,Y 288.583,Z 171.968,A -85,B 0,C 180,E1 -18127.666,E2 -18127.666} C_VEL
LIN {X 0,Y 281.823,Z 158.94,A -85,B 0,C 180,E1 -18129.433,E2 -18129.433} C_VEL
LIN {X 0,Y 275.484,Z 148.08,A -85,B 0,C 180,E1 -18131.185,E2 -18131.185} C_VEL
LIN {X 0,Y 272.043,Z 142.707,A -85,B 0,C 180,E1 -18132.179,E2 -18132.179} C_VEL
LIN {X 0,Y 269.432,Z 138.477,A -85,B 0,C 180,E1 -18132.969,E2 -18132.969} C_VEL
LIN {X 0,Y 266.612,Z 134.033,A -85,B 0,C 180,E1 -18133.849,E2 -18133.849} C_VEL
LIN {X 0,Y 264.336,Z 127.129,A -85,B 0,C 180,E1 -18137.309,E2 -18137.309} C_VEL
LIN {X 0,Y 263.146,Z 123.307,A -85,B 0,C 180,E1 -18139.516,E2 -18139.516} C_VEL
LIN {X 0,Y 263.193,Z 123.319,A -85,B 0,C 180,E1 -18143.237,E2 -18143.237} C_VEL
LIN {X 0,Y 263.144,Z 123.33,A -85,B 0,C 180,E1 -18147.709,E2 -18147.709} C_VEL
LIN {X 0,Y 263.164,Z 123.321,A -85,B 0,C 180,E1 -18151.802,E2 -18151.802} C_VEL
LIN {X 0,Y 263.205,Z 123.316,A -85,B 0,C 180,E1 -18155.215,E2 -18155.215} C_VEL
LIN {X 0,Y 263.278,Z 123.303,A -85,B 0,C 180,E1 -18159.69,E2 -18159.69} C_VEL
LIN {X 0,Y 263.359,Z 123.293,A -85,B 0,C 180,E1 -18164.518,E2 -18164.518} C_VEL
LIN {X 0,Y 263.362,Z 123.297,A -85,B 0,C 180,E1 -18169.229,E2 -18169.229} C_VEL
LIN {X 0,Y 263.538,Z 123.27,A -85,B 0,C 180,E1 -18172.333,E2 -18172.333} C_VEL
LIN {X 0,Y 263.752,Z 123.253,A -85,B 0,C 180,E1 -18178.468,E2 -18178.468} C_VEL
LIN {X 0,Y 263.756,Z 123.243,A -85,B 0,C 180,E1 -18181.522,E2 -18181.522} C_VEL
LIN {X 0,Y 263.538,Z 123.284,A -85,B 0,C 180,E1 -18187.657,E2 -18187.657} C_VEL
LIN {X 0,Y 263.357,Z 123.303,A -85,B 0,C 180,E1 -18190.761,E2 -18190.761} C_VEL
LIN {X 0,Y 263.353,Z 123.305,A -85,B 0,C 180,E1 -18195.472,E2 -18195.472} C_VEL
LIN {X 0,Y 263.264,Z 123.308,A -85,B 0,C 180,E1 -18200.3,E2 -18200.3} C_VEL
LIN {X 0,Y 263.204,Z 123.322,A -85,B 0,C 180,E1 -18205.285,E2 -18205.285} C_VEL
LIN {X 0,Y 263.187,Z 123.392,A -85,B 0,C 180,E1 -18208.631,E2 -18208.631} C_VEL
LIN {X 0,Y 263.55,Z 124.935,A -85,B 0,C 180,E1 -18209.388,E2 -18209.388} C_VEL
LIN {X 0,Y 265.112,Z 127.395,A -85,B 0,C 180,E1 -18209.908,E2 -18209.908} C_VEL
LIN {X 0,Y 267.951,Z 131.099,A -85,B 0,C 180,E1 -18210.789,E2 -18210.789} C_VEL
LIN {X 0,Y 270.665,Z 134.865,A -85,B 0,C 180,E1 -18211.606,E2 -18211.606} C_VEL
LIN {X 0,Y 277.492,Z 145.372,A -85,B 0,C 180,E1 -18213.576,E2 -18213.576} C_VEL
LIN {X 0,Y 284.491,Z 157.042,A -85,B 0,C 180,E1 -18215.456,E2 -18215.456} C_VEL
LIN {X 0,Y 291.498,Z 170.238,A -85,B 0,C 180,E1 -18217.232,E2 -18217.232} C_VEL
LIN {X 0,Y 296.35,Z 180.626,A -85,B 0,C 180,E1 -18218.425,E2 -18218.425} C_VEL
LIN {X 0,Y 292.521,Z 260.388,A -85,B 0,C 180,E1 -18220.386,E2 -18220.386} C_VEL
LIN {X 0,Y 291.082,Z 274.918,A -85,B 0,C 180,E1 -18220.993,E2 -18220.993} C_VEL
LIN {X 0,Y 289.055,Z 289.162,A -85,B 0,C 180,E1 -18221.872,E2 -18221.872} C_VEL
LIN {X 0,Y 286.705,Z 302.522,A -85,B 0,C 180,E1 -18223.006,E2 -18223.006} C_VEL
LIN {X 0,Y 283.943,Z 315.121,A -85,B 0,C 180,E1 -18224.379,E2 -18224.379} C_VEL
LIN {X 0,Y 280.89,Z 326.922,A -85,B 0,C 180,E1 -18225.995,E2 -18225.995} C_VEL
LIN {X 0,Y 277.659,Z 337.913,A -85,B 0,C 180,E1 -18227.872,E2 -18227.872} C_VEL
LIN {X 0,Y 274.812,Z 346.943,A -85,B 0,C 180,E1 -18229.776,E2 -18229.776} C_VEL
LIN {X 0,Y 271.709,Z 355.926,A -85,B 0,C 180,E1 -18232.095,E2 -18232.095} C_VEL
LIN {X 0,Y 269.159,Z 363.062,A -85,B 0,C 180,E1 -18234.374,E2 -18234.374} C_VEL
LIN {X 0,Y 266.571,Z 369.952,A -85,B 0,C 180,E1 -18237.138,E2 -18237.138} C_VEL
LIN {X 0,Y 264.718,Z 374.951,A -85,B 0,C 180,E1 -18239.704,E2 -18239.704} C_VEL
LIN {X 0,Y 263.63,Z 377.843,A -85,B 0,C 180,E1 -18241.596,E2 -18241.596} C_VEL
LIN {X 0,Y 262.291,Z 381.322,A -85,B 0,C 180,E1 -18244.612,E2 -18244.612} C_VEL
LIN {X 0,Y 261.371,Z 383.594,A -85,B 0,C 180,E1 -18247.884,E2 -18247.884} C_VEL
LIN {X 0,Y 260.95,Z 384.395,A -85,B 0,C 180,E1 -18251.142,E2 -18251.142} C_VEL
LIN {X 0,Y 260.788,Z 383.766,A -85,B 0,C 180,E1 -18254.364,E2 -18254.364} C_VEL
LIN {X 0,Y 260.852,Z 382.909,A -85,B 0,C 180,E1 -18255.965,E2 -18255.965} C_VEL
LIN {X 0,Y 261.034,Z 380.129,A -85,B 0,C 180,E1 -18259.135,E2 -18259.135} C_VEL
LIN {X 0,Y 261.462,Z 377.1,A -85,B 0,C 180,E1 -18261.496,E2 -18261.496} C_VEL
LIN {X 0,Y 261.975,Z 373.172,A -85,B 0,C 180,E1 -18263.838,E2 -18263.838} C_VEL
LIN {X 0,Y 262.697,Z 368.329,A -85,B 0,C 180,E1 -18266.163,E2 -18266.163} C_VEL
LIN {X 0,Y 263.929,Z 361.326,A -85,B 0,C 180,E1 -18268.853,E2 -18268.853} C_VEL
LIN {X 0,Y 265.588,Z 352.65,A -85,B 0,C 180,E1 -18271.514,E2 -18271.514} C_VEL
LIN {X 0,Y 267.377,Z 343.263,A -85,B 0,C 180,E1 -18273.841,E2 -18273.841} C_VEL
LIN {X 0,Y 269.328,Z 332.632,A -85,B 0,C 180,E1 -18275.989,E2 -18275.989} C_VEL
LIN {X 0,Y 271.315,Z 321.474,A -85,B 0,C 180,E1 -18277.814,E2 -18277.814} C_VEL
LIN {X 0,Y 273.247,Z 309.165,A -85,B 0,C 180,E1 -18279.435,E2 -18279.435} C_VEL
LIN {X 0,Y 274.85,Z 297.358,A -85,B 0,C 180,E1 -18280.681,E2 -18280.681} C_VEL
LIN {X 0,Y 276.363,Z 284.471,A -85,B 0,C 180,E1 -18281.736,E2 -18281.736} C_VEL
LIN {X 0,Y 277.499,Z 270.8,A -85,B 0,C 180,E1 -18282.569,E2 -18282.569} C_VEL
LIN {X 0,Y 278.318,Z 256.825,A -85,B 0,C 180,E1 -18283.134,E2 -18283.134} C_VEL
LIN {X 0,Y 281.478,Z 167.11,A -85,B 0,C 180,E1 -18285.387,E2 -18285.387} C_VEL
LIN {X 0,Y 274.529,Z 148.752,A -85,B 0,C 180,E1 -18286.649,E2 -18286.649} C_VEL
LIN {X 0,Y 268.554,Z 134.644,A -85,B 0,C 180,E1 -18287.74,E2 -18287.74} C_VEL
LIN {X 0,Y 264.608,Z 126.732,A -85,B 0,C 180,E1 -18288.448,E2 -18288.448} C_VEL
LIN {X 0,Y 263.401,Z 124.272,A -85,B 0,C 180,E1 -18288.671,E2 -18288.671} C_VEL
LIN {X 0,Y 263.217,Z 123.326,A -85,B 0,C 180,E1 -18288.735,E2 -18288.735} C_VEL
LIN {X 0,Y 263.197,Z 123.326,A -85,B 0,C 180,E1 -18291.95,E2 -18291.95} C_VEL
LIN {X 0,Y 263.185,Z 123.328,A -85,B 0,C 180,E1 -18295.291,E2 -18295.291} C_VEL
LIN {X 0,Y 263.147,Z 123.329,A -85,B 0,C 180,E1 -18298.731,E2 -18298.731} C_VEL
LIN {X 0,Y 263.103,Z 123.335,A -85,B 0,C 180,E1 -18302.29,E2 -18302.29} C_VEL
LIN {X 0,Y 263.169,Z 123.326,A -85,B 0,C 180,E1 -18305.978,E2 -18305.978} C_VEL
LIN {X 0,Y 263.182,Z 123.325,A -85,B 0,C 180,E1 -18309.855,E2 -18309.855} C_VEL
LIN {X 0,Y 263.165,Z 123.313,A -85,B 0,C 180,E1 -18313.972,E2 -18313.972} C_VEL
LIN {X 0,Y 263.185,Z 123.326,A -85,B 0,C 180,E1 -18318.388,E2 -18318.388} C_VEL
LIN {X 0,Y 263.18,Z 123.317,A -85,B 0,C 180,E1 -18323.233,E2 -18323.233} C_VEL
LIN {X 0,Y 263.159,Z 123.327,A -85,B 0,C 180,E1 -18325.894,E2 -18325.894} C_VEL
LIN {X 0,Y 263.118,Z 123.326,A -85,B 0,C 180,E1 -18329.51,E2 -18329.51} C_VEL
LIN {X 0,Y 263.174,Z 123.316,A -85,B 0,C 180,E1 -18333.007,E2 -18333.007} C_VEL
LIN {X 0,Y 263.205,Z 123.325,A -85,B 0,C 180,E1 -18336.395,E2 -18336.395} C_VEL
LIN {X 0,Y 263.274,Z 123.312,A -85,B 0,C 180,E1 -18339.7,E2 -18339.7} C_VEL
LIN {X 0,Y 263.33,Z 123.307,A -85,B 0,C 180,E1 -18343.897,E2 -18343.897} C_VEL
LIN {X 0,Y 262.677,Z 123.385,A -85,B 0,C 180,E1 -18345.172,E2 -18345.172} C_VEL
LIN {X 0,Y 259.919,Z 123.732,A -85,B 0,C 180,E1 -18347.253,E2 -18347.253} C_VEL
LIN {X 0,Y 257.577,Z 124.027,A -85,B 0,C 180,E1 -18348.945,E2 -18348.945} C_VEL
LIN {X 0,Y 256.565,Z 124.146,A -85,B 0,C 180,E1 -18350.255,E2 -18350.255} C_VEL
LIN {X 0,Y 256.478,Z 124.153,A -85,B 0,C 180,E1 -18350.698,E2 -18350.698} C_VEL
LIN {X 0,Y 256.476,Z 124.14,A -85,B 0,C 180,E1 -18353.713,E2 -18353.713} C_VEL
LIN {X 0,Y 256.707,Z 124.13,A -85,B 0,C 180,E1 -18358.436,E2 -18358.436} C_VEL
LIN {X 0,Y 256.706,Z 124.127,A -85,B 0,C 180,E1 -18361.574,E2 -18361.574} C_VEL
LIN {X 0,Y 256.532,Z 124.151,A -85,B 0,C 180,E1 -18367.878,E2 -18367.878} C_VEL
LIN {X 0,Y 256.303,Z 124.182,A -85,B 0,C 180,E1 -18371.071,E2 -18371.071} C_VEL
LIN {X 0,Y 256.295,Z 124.182,A -85,B 0,C 180,E1 -18375.92,E2 -18375.92} C_VEL
LIN {X 0,Y 256.164,Z 124.201,A -85,B 0,C 180,E1 -18380.9,E2 -18380.9} C_VEL
LIN {X 0,Y 256.187,Z 124.196,A -85,B 0,C 180,E1 -18385.143,E2 -18385.143} C_VEL
LIN {X 0,Y 256.114,Z 124.203,A -85,B 0,C 180,E1 -18389.604,E2 -18389.604} C_VEL
LIN {X 0,Y 256.068,Z 124.209,A -85,B 0,C 180,E1 -18393.298,E2 -18393.298} C_VEL
LIN {X 0,Y 256.117,Z 124.205,A -85,B 0,C 180,E1 -18397.276,E2 -18397.276} C_VEL
LIN {X 0,Y 256.057,Z 124.207,A -85,B 0,C 180,E1 -18401.208,E2 -18401.208} C_VEL
LIN {X 0,Y 256.045,Z 124.218,A -85,B 0,C 180,E1 -18405.538,E2 -18405.538} C_VEL
LIN {X 0,Y 256.059,Z 124.208,A -85,B 0,C 180,E1 -18408.801,E2 -18408.801} C_VEL
LIN {X 0,Y 256.123,Z 124.393,A -85,B 0,C 180,E1 -18410.87,E2 -18410.87} C_VEL
LIN {X 0,Y 258.673,Z 134.709,A -85,B 0,C 180,E1 -18414.601,E2 -18414.601} C_VEL
LIN {X 0,Y 258.883,Z 135.476,A -85,B 0,C 180,E1 -18414.754,E2 -18414.754} C_VEL
LIN {X 0,Y 268.09,Z 157.479,A -85,B 0,C 180,E1 -18416.529,E2 -18416.529} C_VEL
LIN {X 0,Y 271.458,Z 166.688,A -85,B 0,C 180,E1 -18417.181,E2 -18417.181} C_VEL
LIN {X 0,Y 274.533,Z 188.472,A -85,B 0,C 180,E1 -18418.149,E2 -18418.149} C_VEL
LIN {X 0,Y 271.66,Z 272.938,A -85,B 0,C 180,E1 -18420.348,E2 -18420.348} C_VEL
LIN {X 0,Y 270.583,Z 286.99,A -85,B 0,C 180,E1 -18420.965,E2 -18420.965} C_VEL
LIN {X 0,Y 269.053,Z 300.708,A -85,B 0,C 180,E1 -18421.85,E2 -18421.85} C_VEL
LIN {X 0,Y 267.195,Z 314.054,A -85,B 0,C 180,E1 -18423.02,E2 -18423.02} C_VEL
LIN {X 0,Y 265.396,Z 326.53,A -85,B 0,C 180,E1 -18424.451,E2 -18424.451} C_VEL
LIN {X 0,Y 263.396,Z 337.478,A -85,B 0,C 180,E1 -18425.992,E2 -18425.992} C_VEL
LIN {X 0,Y 261.684,Z 346.416,A -85,B 0,C 180,E1 -18427.501,E2 -18427.501} C_VEL
LIN {X 0,Y 259.514,Z 357.539,A -85,B 0,C 180,E1 -18429.803,E2 -18429.803} C_VEL
LIN {X 0,Y 257.802,Z 366.715,A -85,B 0,C 180,E1 -18432.143,E2 -18432.143} C_VEL
LIN {X 0,Y 256.277,Z 375.471,A -85,B 0,C 180,E1 -18434.901,E2 -18434.901} C_VEL
LIN {X 0,Y 255.231,Z 381.584,A -85,B 0,C 180,E1 -18437.277,E2 -18437.277} C_VEL
LIN {X 0,Y 254.401,Z 388.075,A -85,B 0,C 180,E1 -18440.461,E2 -18440.461} C_VEL
LIN {X 0,Y 254.051,Z 392.883,A -85,B 0,C 180,E1 -18443.649,E2 -18443.649} C_VEL
LIN {X 0,Y 253.987,Z 396.14,A -85,B 0,C 180,E1 -18446.83,E2 -18446.83} C_VEL
LIN {X 0,Y 254.061,Z 397.97,A -85,B 0,C 180,E1 -18450.002,E2 -18450.002} C_VEL
LIN {X 0,Y 254.018,Z 398.373,A -85,B 0,C 180,E1 -18451.588,E2 -18451.588} C_VEL
LIN {X 0,Y 253.935,Z 398.148,A -85,B 0,C 180,E1 -18454.861,E2 -18454.861} C_VEL
LIN {X 0,Y 254.247,Z 396.67,A -85,B 0,C 180,E1 -18457.947,E2 -18457.947} C_VEL
LIN {X 0,Y 254.99,Z 393.822,A -85,B 0,C 180,E1 -18461.126,E2 -18461.126} C_VEL
LIN {X 0,Y 256.381,Z 389.566,A -85,B 0,C 180,E1 -18464.285,E2 -18464.285} C_VEL
LIN {X 0,Y 258.474,Z 383.786,A -85,B 0,C 180,E1 -18467.405,E2 -18467.405} C_VEL
LIN {X 0,Y 260.729,Z 377.317,A -85,B 0,C 180,E1 -18470.103,E2 -18470.103} C_VEL
LIN {X 0,Y 263.69,Z 369.325,A -85,B 0,C 180,E1 -18472.737,E2 -18472.737} C_VEL
LIN {X 0,Y 267.269,Z 359.457,A -85,B 0,C 180,E1 -18475.299,E2 -18475.299} C_VEL
LIN {X 0,Y 270.76,Z 349.098,A -85,B 0,C 180,E1 -18477.436,E2 -18477.436} C_VEL
LIN {X 0,Y 273.903,Z 338.719,A -85,B 0,C 180,E1 -18479.18,E2 -18479.18} C_VEL
LIN {X 0,Y 276.997,Z 327.465,A -85,B 0,C 180,E1 -18480.707,E2 -18480.707} C_VEL
LIN {X 0,Y 279.952,Z 315.194,A -85,B 0,C 180,E1 -18482.03,E2 -18482.03} C_VEL
LIN {X 0,Y 282.678,Z 301.561,A -85,B 0,C 180,E1 -18483.161,E2 -18483.161} C_VEL
LIN {X 0,Y 285.005,Z 287.194,A -85,B 0,C 180,E1 -18484.02,E2 -18484.02} C_VEL
LIN {X 0,Y 286.604,Z 272.916,A -85,B 0,C 180,E1 -18484.599,E2 -18484.599} C_VEL
LIN {X 0,Y 289.731,Z 209.603,A -85,B 0,C 180,E1 -18486.195,E2 -18486.195} C_VEL
LIN {X 0,Y 290.442,Z 193.892,A -85,B 0,C 180,E1 -18486.591,E2 -18486.591} C_VEL
LIN {X 0,Y 289.351,Z 187.864,A -85,B 0,C 180,E1 -18486.988,E2 -18486.988} C_VEL
LIN {X 0,Y 283.504,Z 175.001,A -85,B 0,C 180,E1 -18488.528,E2 -18488.528} C_VEL
LIN {X 0,Y 277.314,Z 163.021,A -85,B 0,C 180,E1 -18490.225,E2 -18490.225} C_VEL
LIN {X 0,Y 271.304,Z 152.533,A -85,B 0,C 180,E1 -18491.963,E2 -18491.963} C_VEL
LIN {X 0,Y 265.596,Z 143.468,A -85,B 0,C 180,E1 -18493.713,E2 -18493.713} C_VEL
LIN {X 0,Y 262.233,Z 138.366,A -85,B 0,C 180,E1 -18494.806,E2 -18494.806} C_VEL
LIN {X 0,Y 259.313,Z 133.95,A -85,B 0,C 180,E1 -18495.805,E2 -18495.805} C_VEL
LIN {X 0,Y 259.021,Z 133.338,A -85,B 0,C 180,E1 -18495.945,E2 -18495.945} C_VEL
LIN {X 0,Y 257.242,Z 127.796,A -85,B 0,C 180,E1 -18499.023,E2 -18499.023} C_VEL
LIN {X 0,Y 256.11,Z 124.209,A -85,B 0,C 180,E1 -18501.239,E2 -18501.239} C_VEL
LIN {X 0,Y 256.122,Z 124.199,A -85,B 0,C 180,E1 -18505.41,E2 -18505.41} C_VEL
LIN {X 0,Y 256.099,Z 124.201,A -85,B 0,C 180,E1 -18508.568,E2 -18508.568} C_VEL
LIN {X 0,Y 256.109,Z 124.198,A -85,B 0,C 180,E1 -18512.188,E2 -18512.188} C_VEL
LIN {X 0,Y 256.149,Z 124.192,A -85,B 0,C 180,E1 -18515.693,E2 -18515.693} C_VEL
LIN {X 0,Y 256.177,Z 124.19,A -85,B 0,C 180,E1 -18519.101,E2 -18519.101} C_VEL
LIN {X 0,Y 256.294,Z 124.172,A -85,B 0,C 180,E1 -18524.08,E2 -18524.08} C_VEL
LIN {X 0,Y 256.304,Z 124.173,A -85,B 0,C 180,E1 -18528.929,E2 -18528.929} C_VEL
LIN {X 0,Y 256.48,Z 124.15,A -85,B 0,C 180,E1 -18532.12,E2 -18532.12} C_VEL
LIN {X 0,Y 256.473,Z 124.149,A -85,B 0,C 180,E1 -18536.853,E2 -18536.853} C_VEL
LIN {X 0,Y 256.758,Z 124.121,A -85,B 0,C 180,E1 -18539.995,E2 -18539.995} C_VEL
LIN {X 0,Y 256.498,Z 124.16,A -85,B 0,C 180,E1 -18543.136,E2 -18543.136} C_VEL
LIN {X 0,Y 256.5,Z 124.158,A -85,B 0,C 180,E1 -18547.869,E2 -18547.869} C_VEL
LIN {X 0,Y 256.296,Z 124.176,A -85,B 0,C 180,E1 -18552.666,E2 -18552.666} C_VEL
LIN {X 0,Y 256.284,Z 124.178,A -85,B 0,C 180,E1 -18556.296,E2 -18556.296} C_VEL
LIN {X 0,Y 256.158,Z 124.198,A -85,B 0,C 180,E1 -18561.115,E2 -18561.115} C_VEL
LIN {X 0,Y 256.184,Z 124.197,A -85,B 0,C 180,E1 -18565.132,E2 -18565.132} C_VEL
LIN {X 0,Y 256.167,Z 124.283,A -85,B 0,C 180,E1 -18566.909,E2 -18566.909} C_VEL
LIN {X 0,Y 256.306,Z 125.049,A -85,B 0,C 180,E1 -18567.334,E2 -18567.334} C_VEL
LIN {X 0,Y 257.481,Z 127.542,A -85,B 0,C 180,E1 -18567.798,E2 -18567.798} C_VEL
LIN {X 0,Y 260.231,Z 130.593,A -85,B 0,C 180,E1 -18568.725,E2 -18568.725} C_VEL
LIN {X 0,Y 263.553,Z 135.146,A -85,B 0,C 180,E1 -18569.827,E2 -18569.827} C_VEL
LIN {X 0,Y 268.887,Z 143.102,A -85,B 0,C 180,E1 -18571.51,E2 -18571.51} C_VEL
LIN {X 0,Y 273.366,Z 149.892,A -85,B 0,C 180,E1 -18572.831,E2 -18572.831} C_VEL
LIN {X 0,Y 280.427,Z 161.898,A -85,B 0,C 180,E1 -18574.809,E2 -18574.809} C_VEL
LIN {X 0,Y 287.364,Z 175.251,A -85,B 0,C 180,E1 -18576.641,E2 -18576.641} C_VEL
LIN {X 0,Y 290.984,Z 183.177,A -85,B 0,C 180,E1 -18577.571,E2 -18577.571} C_VEL
LIN {X 0,Y 287.071,Z 260.388,A -85,B 0,C 180,E1 -18579.486,E2 -18579.486} C_VEL
LIN {X 0,Y 285.613,Z 274.778,A -85,B 0,C 180,E1 -18580.089,E2 -18580.089} C_VEL
LIN {X 0,Y 283.679,Z 288.225,A -85,B 0,C 180,E1 -18580.918,E2 -18580.918} C_VEL
LIN {X 0,Y 281.449,Z 300.586,A -85,B 0,C 180,E1 -18581.941,E2 -18581.941} C_VEL
LIN {X 0,Y 278.705,Z 313.059,A -85,B 0,C 180,E1 -18583.268,E2 -18583.268} C_VEL
LIN {X 0,Y 275.414,Z 325.398,A -85,B 0,C 180,E1 -18584.916,E2 -18584.916} C_VEL
LIN {X 0,Y 272.092,Z 336.588,A -85,B 0,C 180,E1 -18586.803,E2 -18586.803} C_VEL
LIN {X 0,Y 269.03,Z 345.848,A -85,B 0,C 180,E1 -18588.727,E2 -18588.727} C_VEL
LIN {X 0,Y 265.742,Z 355.081,A -85,B 0,C 180,E1 -18591.087,E2 -18591.087} C_VEL
LIN {X 0,Y 263.178,Z 361.865,A -85,B 0,C 180,E1 -18593.227,E2 -18593.227} C_VEL
LIN {X 0,Y 260.788,Z 367.881,A -85,B 0,C 180,E1 -18595.531,E2 -18595.531} C_VEL
LIN {X 0,Y 258.761,Z 373.102,A -85,B 0,C 180,E1 -18598.018,E2 -18598.018} C_VEL
LIN {X 0,Y 256.752,Z 378.086,A -85,B 0,C 180,E1 -18601.14,E2 -18601.14} C_VEL
LIN {X 0,Y 255.456,Z 381.232,A -85,B 0,C 180,E1 -18603.882,E2 -18603.882} C_VEL
LIN {X 0,Y 254.896,Z 382.623,A -85,B 0,C 180,E1 -18605.568,E2 -18605.568} C_VEL
LIN {X 0,Y 254.086,Z 384.283,A -85,B 0,C 180,E1 -18608.923,E2 -18608.923} C_VEL
LIN {X 0,Y 253.916,Z 384.565,A -85,B 0,C 180,E1 -18610.599,E2 -18610.599} C_VEL
LIN {X 0,Y 253.686,Z 384.066,A -85,B 0,C 180,E1 -18613.914,E2 -18613.914} C_VEL
LIN {X 0,Y 253.723,Z 383.17,A -85,B 0,C 180,E1 -18615.779,E2 -18615.779} C_VEL
LIN {X 0,Y 253.895,Z 380.672,A -85,B 0,C 180,E1 -18618.825,E2 -18618.825} C_VEL
LIN {X 0,Y 254.336,Z 377.709,A -85,B 0,C 180,E1 -18621.256,E2 -18621.256} C_VEL
LIN {X 0,Y 254.833,Z 373.917,A -85,B 0,C 180,E1 -18623.664,E2 -18623.664} C_VEL
LIN {X 0,Y 255.555,Z 369.218,A -85,B 0,C 180,E1 -18626.055,E2 -18626.055} C_VEL
LIN {X 0,Y 256.769,Z 362.379,A -85,B 0,C 180,E1 -18628.822,E2 -18628.822} C_VEL
LIN {X 0,Y 258.208,Z 355.237,A -85,B 0,C 180,E1 -18631.167,E2 -18631.167} C_VEL
LIN {X 0,Y 259.953,Z 346.491,A -85,B 0,C 180,E1 -18633.524,E2 -18633.524} C_VEL
LIN {X 0,Y 262.031,Z 335.881,A -85,B 0,C 180,E1 -18635.843,E2 -18635.843} C_VEL
LIN {X 0,Y 263.789,Z 325.836,A -85,B 0,C 180,E1 -18637.653,E2 -18637.653} C_VEL
LIN {X 0,Y 265.851,Z 314.444,A -85,B 0,C 180,E1 -18639.316,E2 -18639.316} C_VEL
LIN {X 0,Y 267.692,Z 302.046,A -85,B 0,C 180,E1 -18640.779,E2 -18640.779} C_VEL
LIN {X 0,Y 269.443,Z 288.204,A -85,B 0,C 180,E1 -18642.042,E2 -18642.042} C_VEL
LIN {X 0,Y 270.747,Z 274.337,A -85,B 0,C 180,E1 -18642.983,E2 -18642.983} C_VEL
LIN {X 0,Y 271.692,Z 259.92,A -85,B 0,C 180,E1 -18643.651,E2 -18643.651} C_VEL
LIN {X 0,Y 275.06,Z 168.977,A -85,B 0,C 180,E1 -18645.999,E2 -18645.999} C_VEL
LIN {X 0,Y 270.741,Z 156.915,A -85,B 0,C 180,E1 -18646.822,E2 -18646.822} C_VEL
LIN {X 0,Y 263.883,Z 140.149,A -85,B 0,C 180,E1 -18648.12,E2 -18648.12} C_VEL
LIN {X 0,Y 259.266,Z 130.76,A -85,B 0,C 180,E1 -18648.98,E2 -18648.98} C_VEL
LIN {X 0,Y 256.467,Z 125.377,A -85,B 0,C 180,E1 -18649.511,E2 -18649.511} C_VEL
LIN {X 0,Y 256.24,Z 124.217,A -85,B 0,C 180,E1 -18649.578,E2 -18649.578} C_VEL
LIN {X 0,Y 256.156,Z 124.201,A -85,B 0,C 180,E1 -18654.299,E2 -18654.299} C_VEL
LIN {X 0,Y 256.106,Z 124.206,A -85,B 0,C 180,E1 -18658.596,E2 -18658.596} C_VEL
LIN {X 0,Y 256.054,Z 124.215,A -85,B 0,C 180,E1 -18663.292,E2 -18663.292} C_VEL
LIN {X 0,Y 256.13,Z 124.205,A -85,B 0,C 180,E1 -18667.286,E2 -18667.286} C_VEL
LIN {X 0,Y 256.14,Z 124.201,A -85,B 0,C 180,E1 -18671.183,E2 -18671.183} C_VEL
LIN {X 0,Y 256.09,Z 124.204,A -85,B 0,C 180,E1 -18675.519,E2 -18675.519} C_VEL
LIN {X 0,Y 256.105,Z 124.204,A -85,B 0,C 180,E1 -18678.815,E2 -18678.815} C_VEL
LIN {X 0,Y 256.13,Z 124.191,A -85,B 0,C 180,E1 -18682.875,E2 -18682.875} C_VEL
LIN {X 0,Y 256.061,Z 124.212,A -85,B 0,C 180,E1 -18686.714,E2 -18686.714} C_VEL
LIN {X 0,Y 256.104,Z 124.185,A -85,B 0,C 180,E1 -18691.414,E2 -18691.414} C_VEL
LIN {X 0,Y 256.169,Z 124.198,A -85,B 0,C 180,E1 -18695.706,E2 -18695.706} C_VEL
LIN {X 0,Y 256.223,Z 124.189,A -85,B 0,C 180,E1 -18699.116,E2 -18699.116} C_VEL
LIN {X 0,Y 256.283,Z 124.183,A -85,B 0,C 180,E1 -18704.09,E2 -18704.09} C_VEL
LIN {X 0,Y 256.295,Z 124.182,A -85,B 0,C 180,E1 -18708.939,E2 -18708.939} C_VEL
LIN {X 0,Y 256.478,Z 124.153,A -85,B 0,C 180,E1 -18710.698,E2 -18710.698} C_VEL
LIN {X 0,Y 255.775,Z 124.234,A -85,B 0,C 180,E1 -18712.008,E2 -18712.008} C_VEL
LIN {X 0,Y 252.861,Z 124.59,A -85,B 0,C 180,E1 -18714.142,E2 -18714.142} C_VEL
LIN {X 0,Y 250.474,Z 124.898,A -85,B 0,C 180,E1 -18715.88,E2 -18715.88} C_VEL
LIN {X 0,Y 249.558,Z 125.018,A -85,B 0,C 180,E1 -18717.228,E2 -18717.228} C_VEL
LIN {X 0,Y 249.54,Z 125.017,A -85,B 0,C 180,E1 -18717.683,E2 -18717.683} C_VEL
LIN {X 0,Y 249.726,Z 125,A -85,B 0,C 180,E1 -18720.005,E2 -18720.005} C_VEL
LIN {X 0,Y 249.427,Z 125.022,A -85,B 0,C 180,E1 -18723.236,E2 -18723.236} C_VEL
LIN {X 0,Y 249.474,Z 125.03,A -85,B 0,C 180,E1 -18728.102,E2 -18728.102} C_VEL
LIN {X 0,Y 249.247,Z 125.059,A -85,B 0,C 180,E1 -18731.389,E2 -18731.389} C_VEL
LIN {X 0,Y 249.238,Z 125.063,A -85,B 0,C 180,E1 -18736.383,E2 -18736.383} C_VEL
LIN {X 0,Y 249.084,Z 125.081,A -85,B 0,C 180,E1 -18741.523,E2 -18741.523} C_VEL
LIN {X 0,Y 249.129,Z 125.075,A -85,B 0,C 180,E1 -18745.487,E2 -18745.487} C_VEL
LIN {X 0,Y 249.083,Z 125.08,A -85,B 0,C 180,E1 -18748.998,E2 -18748.998} C_VEL
LIN {X 0,Y 249.031,Z 125.084,A -85,B 0,C 180,E1 -18752.431,E2 -18752.431} C_VEL
LIN {X 0,Y 249.05,Z 125.088,A -85,B 0,C 180,E1 -18756.347,E2 -18756.347} C_VEL
LIN {X 0,Y 248.994,Z 125.084,A -85,B 0,C 180,E1 -18760.486,E2 -18760.486} C_VEL
LIN {X 0,Y 249.004,Z 125.093,A -85,B 0,C 180,E1 -18762.795,E2 -18762.795} C_VEL
LIN {X 0,Y 249.014,Z 125.093,A -85,B 0,C 180,E1 -18767.366,E2 -18767.366} C_VEL
LIN {X 0,Y 249.027,Z 125.164,A -85,B 0,C 180,E1 -18770.129,E2 -18770.129} C_VEL
LIN {X 0,Y 251.475,Z 134.849,A -85,B 0,C 180,E1 -18773.775,E2 -18773.775} C_VEL
LIN {X 0,Y 261.419,Z 158.325,A -85,B 0,C 180,E1 -18775.781,E2 -18775.781} C_VEL
LIN {X 0,Y 265.38,Z 169.344,A -85,B 0,C 180,E1 -18776.582,E2 -18776.582} C_VEL
LIN {X 0,Y 268.139,Z 190.4,A -85,B 0,C 180,E1 -18777.526,E2 -18777.526} C_VEL
LIN {X 0,Y 265.226,Z 272.728,A -85,B 0,C 180,E1 -18779.718,E2 -18779.718} C_VEL
LIN {X 0,Y 264.089,Z 286.78,A -85,B 0,C 180,E1 -18780.345,E2 -18780.345} C_VEL
LIN {X 0,Y 262.635,Z 299.951,A -85,B 0,C 180,E1 -18781.208,E2 -18781.208} C_VEL
LIN {X 0,Y 260.878,Z 312.536,A -85,B 0,C 180,E1 -18782.311,E2 -18782.311} C_VEL
LIN {X 0,Y 259.041,Z 324.739,A -85,B 0,C 180,E1 -18783.699,E2 -18783.699} C_VEL
LIN {X 0,Y 256.822,Z 336.396,A -85,B 0,C 180,E1 -18785.337,E2 -18785.337} C_VEL
LIN {X 0,Y 255.131,Z 345.468,A -85,B 0,C 180,E1 -18786.89,E2 -18786.89} C_VEL
LIN {X 0,Y 253.156,Z 355.021,A -85,B 0,C 180,E1 -18788.847,E2 -18788.847} C_VEL
LIN {X 0,Y 251.235,Z 364.62,A -85,B 0,C 180,E1 -18791.237,E2 -18791.237} C_VEL
LIN {X 0,Y 249.629,Z 373.738,A -85,B 0,C 180,E1 -18794.07,E2 -18794.07} C_VEL
LIN {X 0,Y 248.269,Z 381.06,A -85,B 0,C 180,E1 -18796.913,E2 -18796.913} C_VEL
LIN {X 0,Y 247.531,Z 386.175,A -85,B 0,C 180,E1 -18799.367,E2 -18799.367} C_VEL
LIN {X 0,Y 247.136,Z 390.26,A -85,B 0,C 180,E1 -18801.828,E2 -18801.828} C_VEL
LIN {X 0,Y 246.895,Z 394.348,A -85,B 0,C 180,E1 -18805.104,E2 -18805.104} C_VEL
LIN {X 0,Y 246.938,Z 396.956,A -85,B 0,C 180,E1 -18808.371,E2 -18808.371} C_VEL
LIN {X 0,Y 246.99,Z 397.732,A -85,B 0,C 180,E1 -18810.002,E2 -18810.002} C_VEL
LIN {X 0,Y 246.85,Z 398.259,A -85,B 0,C 180,E1 -18813.267,E2 -18813.267} C_VEL
LIN {X 0,Y 246.984,Z 397.465,A -85,B 0,C 180,E1 -18816.538,E2 -18816.538} C_VEL
LIN {X 0,Y 247.536,Z 395.354,A -85,B 0,C 180,E1 -18819.81,E2 -18819.81} C_VEL
LIN {X 0,Y 248.579,Z 391.88,A -85,B 0,C 180,E1 -18823.075,E2 -18823.075} C_VEL
LIN {X 0,Y 250.475,Z 386.947,A -85,B 0,C 180,E1 -18826.298,E2 -18826.298} C_VEL
LIN {X 0,Y 252.968,Z 380.418,A -85,B 0,C 180,E1 -18829.477,E2 -18829.477} C_VEL
LIN {X 0,Y 255.779,Z 373.192,A -85,B 0,C 180,E1 -18832.2,E2 -18832.2} C_VEL
LIN {X 0,Y 258.701,Z 365.652,A -85,B 0,C 180,E1 -18834.477,E2 -18834.477} C_VEL
LIN {X 0,Y 262.03,Z 356.638,A -85,B 0,C 180,E1 -18836.698,E2 -18836.698} C_VEL
LIN {X 0,Y 265.696,Z 346.1,A -85,B 0,C 180,E1 -18838.792,E2 -18838.792} C_VEL
LIN {X 0,Y 269.02,Z 335.237,A -85,B 0,C 180,E1 -18840.541,E2 -18840.541} C_VEL
LIN {X 0,Y 272.158,Z 324.129,A -85,B 0,C 180,E1 -18841.966,E2 -18841.966} C_VEL
LIN {X 0,Y 275.18,Z 311.137,A -85,B 0,C 180,E1 -18843.308,E2 -18843.308} C_VEL
LIN {X 0,Y 277.934,Z 297.417,A -85,B 0,C 180,E1 -18844.349,E2 -18844.349} C_VEL
LIN {X 0,Y 280.08,Z 282.984,A -85,B 0,C 180,E1 -18845.142,E2 -18845.142} C_VEL
LIN {X 0,Y 281.457,Z 268.191,A -85,B 0,C 180,E1 -18845.68,E2 -18845.68} C_VEL
LIN {X 0,Y 285.131,Z 195.267,A -85,B 0,C 180,E1 -18847.512,E2 -18847.512} C_VEL
LIN {X 0,Y 284.365,Z 191.038,A -85,B 0,C 180,E1 -18847.803,E2 -18847.803} C_VEL
LIN {X 0,Y 278.581,Z 178.324,A -85,B 0,C 180,E1 -18849.396,E2 -18849.396} C_VEL
LIN {X 0,Y 273.406,Z 168.032,A -85,B 0,C 180,E1 -18850.886,E2 -18850.886} C_VEL
LIN {X 0,Y 267.053,Z 156.81,A -85,B 0,C 180,E1 -18852.802,E2 -18852.802} C_VEL
LIN {X 0,Y 261.853,Z 148.433,A -85,B 0,C 180,E1 -18854.474,E2 -18854.474} C_VEL
LIN {X 0,Y 258.697,Z 143.586,A -85,B 0,C 180,E1 -18855.545,E2 -18855.545} C_VEL
LIN {X 0,Y 254.987,Z 138.114,A -85,B 0,C 180,E1 -18856.869,E2 -18856.869} C_VEL
LIN {X 0,Y 251.897,Z 133.519,A -85,B 0,C 180,E1 -18858.037,E2 -18858.037} C_VEL
LIN {X 0,Y 251.616,Z 132.911,A -85,B 0,C 180,E1 -18858.218,E2 -18858.218} C_VEL
LIN {X 0,Y 249.094,Z 125.075,A -85,B 0,C 180,E1 -18863.145,E2 -18863.145} C_VEL
LIN {X 0,Y 249.05,Z 125.084,A -85,B 0,C 180,E1 -18867.845,E2 -18867.845} C_VEL
LIN {X 0,Y 249.065,Z 125.081,A -85,B 0,C 180,E1 -18871.329,E2 -18871.329} C_VEL
LIN {X 0,Y 249.118,Z 125.073,A -85,B 0,C 180,E1 -18874.96,E2 -18874.96} C_VEL
LIN {X 0,Y 249.109,Z 125.076,A -85,B 0,C 180,E1 -18878.599,E2 -18878.599} C_VEL
LIN {X 0,Y 249.238,Z 125.052,A -85,B 0,C 180,E1 -18883.617,E2 -18883.617} C_VEL
LIN {X 0,Y 249.248,Z 125.05,A -85,B 0,C 180,E1 -18888.611,E2 -18888.611} C_VEL
LIN {X 0,Y 249.43,Z 125.029,A -85,B 0,C 180,E1 -18891.896,E2 -18891.896} C_VEL
LIN {X 0,Y 249.283,Z 125.058,A -85,B 0,C 180,E1 -18895.143,E2 -18895.143} C_VEL
LIN {X 0,Y 249.675,Z 125.005,A -85,B 0,C 180,E1 -18898.382,E2 -18898.382} C_VEL
LIN {X 0,Y 249.68,Z 124.996,A -85,B 0,C 180,E1 -18901.608,E2 -18901.608} C_VEL
LIN {X 0,Y 249.436,Z 125.032,A -85,B 0,C 180,E1 -18906.568,E2 -18906.568} C_VEL
LIN {X 0,Y 249.348,Z 125.039,A -85,B 0,C 180,E1 -18909.731,E2 -18909.731} C_VEL
LIN {X 0,Y 249.207,Z 125.067,A -85,B 0,C 180,E1 -18914.697,E2 -18914.697} C_VEL
LIN {X 0,Y 249.14,Z 125.074,A -85,B 0,C 180,E1 -18918.071,E2 -18918.071} C_VEL
LIN {X 0,Y 249.087,Z 125.083,A -85,B 0,C 180,E1 -18921.512,E2 -18921.512} C_VEL
LIN {X 0,Y 249.155,Z 125.233,A -85,B 0,C 180,E1 -18925.024,E2 -18925.024} C_VEL
LIN {X 0,Y 250.313,Z 128.243,A -85,B 0,C 180,E1 -18925.617,E2 -18925.617} C_VEL
LIN {X 0,Y 252.544,Z 130.322,A -85,B 0,C 180,E1 -18926.433,E2 -18926.433} C_VEL
LIN {X 0,Y 253.123,Z 130.979,A -85,B 0,C 180,E1 -18926.646,E2 -18926.646} C_VEL
LIN {X 0,Y 255.144,Z 134.149,A -85,B 0,C 180,E1 -18927.414,E2 -18927.414} C_VEL
LIN {X 0,Y 256.91,Z 136.06,A -85,B 0,C 180,E1 -18928.024,E2 -18928.024} C_VEL
LIN {X 0,Y 261.374,Z 142.442,A -85,B 0,C 180,E1 -18929.561,E2 -18929.561} C_VEL
LIN {X 0,Y 267.891,Z 152.283,A -85,B 0,C 180,E1 -18931.64,E2 -18931.64} C_VEL
LIN {X 0,Y 274.298,Z 163.05,A -85,B 0,C 180,E1 -18933.543,E2 -18933.543} C_VEL
LIN {X 0,Y 280.781,Z 175.154,A -85,B 0,C 180,E1 -18935.361,E2 -18935.361} C_VEL
LIN {X 0,Y 285.595,Z 185.313,A -85,B 0,C 180,E1 -18936.654,E2 -18936.654} C_VEL
LIN {X 0,Y 281.623,Z 261.295,A -85,B 0,C 180,E1 -18938.581,E2 -18938.581} C_VEL
LIN {X 0,Y 280.063,Z 275.819,A -85,B 0,C 180,E1 -18939.211,E2 -18939.211} C_VEL
LIN {X 0,Y 277.94,Z 289.727,A -85,B 0,C 180,E1 -18940.099,E2 -18940.099} C_VEL
LIN {X 0,Y 275.521,Z 302.368,A -85,B 0,C 180,E1 -18941.192,E2 -18941.192} C_VEL
LIN {X 0,Y 272.4,Z 315.582,A -85,B 0,C 180,E1 -18942.664,E2 -18942.664} C_VEL
LIN {X 0,Y 269.034,Z 327.497,A -85,B 0,C 180,E1 -18944.344,E2 -18944.344} C_VEL
LIN {X 0,Y 265.842,Z 337.572,A -85,B 0,C 180,E1 -18946.117,E2 -18946.117} C_VEL
LIN {X 0,Y 262.742,Z 346.479,A -85,B 0,C 180,E1 -18948.029,E2 -18948.029} C_VEL
LIN {X 0,Y 259.317,Z 355.636,A -85,B 0,C 180,E1 -18950.437,E2 -18950.437} C_VEL
LIN {X 0,Y 256.319,Z 363.139,A -85,B 0,C 180,E1 -18952.897,E2 -18952.897} C_VEL
LIN {X 0,Y 253.729,Z 369.268,A -85,B 0,C 180,E1 -18955.399,E2 -18955.399} C_VEL
LIN {X 0,Y 251.645,Z 374.232,A -85,B 0,C 180,E1 -18957.949,E2 -18957.949} C_VEL
LIN {X 0,Y 249.908,Z 378.325,A -85,B 0,C 180,E1 -18960.653,E2 -18960.653} C_VEL
LIN {X 0,Y 248.664,Z 381.147,A -85,B 0,C 180,E1 -18963.112,E2 -18963.112} C_VEL
LIN {X 0,Y 247.482,Z 383.683,A -85,B 0,C 180,E1 -18966.571,E2 -18966.571} C_VEL
LIN {X 0,Y 246.877,Z 384.737,A -85,B 0,C 180,E1 -18970.023,E2 -18970.023} C_VEL
LIN {X 0,Y 246.598,Z 384.362,A -85,B 0,C 180,E1 -18973.439,E2 -18973.439} C_VEL
LIN {X 0,Y 246.64,Z 383.398,A -85,B 0,C 180,E1 -18975.627,E2 -18975.627} C_VEL
LIN {X 0,Y 246.768,Z 381.162,A -85,B 0,C 180,E1 -18978.498,E2 -18978.498} C_VEL
LIN {X 0,Y 247.352,Z 377.221,A -85,B 0,C 180,E1 -18981.83,E2 -18981.83} C_VEL
LIN {X 0,Y 247.913,Z 373.213,A -85,B 0,C 180,E1 -18984.303,E2 -18984.303} C_VEL
LIN {X 0,Y 248.709,Z 368.276,A -85,B 0,C 180,E1 -18986.758,E2 -18986.758} C_VEL
LIN {X 0,Y 250.068,Z 361.17,A -85,B 0,C 180,E1 -18989.595,E2 -18989.595} C_VEL
LIN {X 0,Y 251.882,Z 352.376,A -85,B 0,C 180,E1 -18992.396,E2 -18992.396} C_VEL
LIN {X 0,Y 253.881,Z 342.853,A -85,B 0,C 180,E1 -18994.838,E2 -18994.838} C_VEL
LIN {X 0,Y 255.579,Z 334.012,A -85,B 0,C 180,E1 -18996.709,E2 -18996.709} C_VEL
LIN {X 0,Y 257.435,Z 324.243,A -85,B 0,C 180,E1 -18998.436,E2 -18998.436} C_VEL
LIN {X 0,Y 259.513,Z 312.492,A -85,B 0,C 180,E1 -19000.136,E2 -19000.136} C_VEL
LIN {X 0,Y 261.473,Z 299.57,A -85,B 0,C 180,E1 -19001.628,E2 -19001.628} C_VEL
LIN {X 0,Y 263.174,Z 286.109,A -85,B 0,C 180,E1 -19002.823,E2 -19002.823} C_VEL
LIN {X 0,Y 264.48,Z 272.073,A -85,B 0,C 180,E1 -19003.736,E2 -19003.736} C_VEL
LIN {X 0,Y 265.309,Z 258.715,A -85,B 0,C 180,E1 -19004.328,E2 -19004.328} C_VEL
LIN {X 0,Y 268.715,Z 170.652,A -85,B 0,C 180,E1 -19006.635,E2 -19006.635} C_VEL
LIN {X 0,Y 263.859,Z 157.304,A -85,B 0,C 180,E1 -19007.593,E2 -19007.593} C_VEL
LIN {X 0,Y 257.269,Z 141.454,A -85,B 0,C 180,E1 -19008.891,E2 -19008.891} C_VEL
LIN {X 0,Y 251.683,Z 130.587,A -85,B 0,C 180,E1 -19009.975,E2 -19009.975} C_VEL
LIN {X 0,Y 249.323,Z 125.92,A -85,B 0,C 180,E1 -19010.451,E2 -19010.451} C_VEL
LIN {X 0,Y 249.161,Z 125.074,A -85,B 0,C 180,E1 -19010.569,E2 -19010.569} C_VEL
LIN {X 0,Y 249.106,Z 125.082,A -85,B 0,C 180,E1 -19015.486,E2 -19015.486} C_VEL
LIN {X 0,Y 249.051,Z 125.086,A -85,B 0,C 180,E1 -19018.994,E2 -19018.994} C_VEL
LIN {X 0,Y 249.005,Z 125.092,A -85,B 0,C 180,E1 -19022.427,E2 -19022.427} C_VEL
LIN {X 0,Y 249.056,Z 125.085,A -85,B 0,C 180,E1 -19026.338,E2 -19026.338} C_VEL
LIN {X 0,Y 249.107,Z 125.08,A -85,B 0,C 180,E1 -19030.455,E2 -19030.455} C_VEL
LIN {X 0,Y 249.036,Z 125.077,A -85,B 0,C 180,E1 -19034.868,E2 -19034.868} C_VEL
LIN {X 0,Y 249.071,Z 125.082,A -85,B 0,C 180,E1 -19037.384,E2 -19037.384} C_VEL
LIN {X 0,Y 249.027,Z 125.069,A -85,B 0,C 180,E1 -19041.628,E2 -19041.628} C_VEL
LIN {X 0,Y 249.037,Z 125.085,A -85,B 0,C 180,E1 -19045.646,E2 -19045.646} C_VEL
LIN {X 0,Y 249.025,Z 125.08,A -85,B 0,C 180,E1 -19049.477,E2 -19049.477} C_VEL
LIN {X 0,Y 249.054,Z 125.073,A -85,B 0,C 180,E1 -19053.167,E2 -19053.167} C_VEL
LIN {X 0,Y 249.098,Z 125.08,A -85,B 0,C 180,E1 -19056.741,E2 -19056.741} C_VEL
LIN {X 0,Y 249.133,Z 125.073,A -85,B 0,C 180,E1 -19060.22,E2 -19060.22} C_VEL
LIN {X 0,Y 249.225,Z 125.066,A -85,B 0,C 180,E1 -19063.627,E2 -19063.627} C_VEL
LIN {X 0,Y 249.238,Z 125.061,A -85,B 0,C 180,E1 -19068.622,E2 -19068.622} C_VEL
LIN {X 0,Y 249.47,Z 125.018,A -85,B 0,C 180,E1 -19071.908,E2 -19071.908} C_VEL
LIN {X 0,Y 249.431,Z 125.031,A -85,B 0,C 180,E1 -19076.775,E2 -19076.775} C_VEL
LIN {X 0,Y 249.54,Z 125.017,A -85,B 0,C 180,E1 -19077.683,E2 -19077.683} C_VEL
LIN {X 0,Y 248.993,Z 125.093,A -85,B 0,C 180,E1 -19079.031,E2 -19079.031} C_VEL
LIN {X 0,Y 247.399,Z 125.292,A -85,B 0,C 180,E1 -19080.353,E2 -19080.353} C_VEL
LIN {X 0,Y 243.476,Z 125.765,A -85,B 0,C 180,E1 -19083.011,E2 -19083.011} C_VEL
LIN {X 0,Y 242.348,Z 125.897,A -85,B 0,C 180,E1 -19084.402,E2 -19084.402} C_VEL
LIN {X 0,Y 242.253,Z 125.909,A -85,B 0,C 180,E1 -19084.875,E2 -19084.875} C_VEL
LIN {X 0,Y 242.421,Z 125.909,A -85,B 0,C 180,E1 -19088.34,E2 -19088.34} C_VEL
LIN {X 0,Y 242.161,Z 125.944,A -85,B 0,C 180,E1 -19093.43,E2 -19093.43} C_VEL
LIN {X 0,Y 242.146,Z 125.944,A -85,B 0,C 180,E1 -19096.877,E2 -19096.877} C_VEL
LIN {X 0,Y 242.051,Z 125.957,A -85,B 0,C 180,E1 -19101.708,E2 -19101.708} C_VEL
LIN {X 0,Y 242.066,Z 125.955,A -85,B 0,C 180,E1 -19105.843,E2 -19105.843} C_VEL
LIN {X 0,Y 242.03,Z 125.957,A -85,B 0,C 180,E1 -19109.585,E2 -19109.585} C_VEL
LIN {X 0,Y 241.982,Z 125.964,A -85,B 0,C 180,E1 -19113.498,E2 -19113.498} C_VEL
LIN {X 0,Y 241.992,Z 125.966,A -85,B 0,C 180,E1 -19117.587,E2 -19117.587} C_VEL
LIN {X 0,Y 241.933,Z 125.97,A -85,B 0,C 180,E1 -19121.929,E2 -19121.929} C_VEL
LIN {X 0,Y 241.93,Z 125.975,A -85,B 0,C 180,E1 -19126.578,E2 -19126.578} C_VEL
LIN {X 0,Y 241.998,Z 126.167,A -85,B 0,C 180,E1 -19129.437,E2 -19129.437} C_VEL
LIN {X 0,Y 244.174,Z 134.565,A -85,B 0,C 180,E1 -19132.737,E2 -19132.737} C_VEL
LIN {X 0,Y 252.684,Z 154.161,A -85,B 0,C 180,E1 -19134.567,E2 -19134.567} C_VEL
LIN {X 0,Y 259.143,Z 170.822,A -85,B 0,C 180,E1 -19135.901,E2 -19135.901} C_VEL
LIN {X 0,Y 261.804,Z 190.929,A -85,B 0,C 180,E1 -19136.837,E2 -19136.837} C_VEL
LIN {X 0,Y 258.82,Z 272.49,A -85,B 0,C 180,E1 -19139.057,E2 -19139.057} C_VEL
LIN {X 0,Y 257.608,Z 286.544,A -85,B 0,C 180,E1 -19139.691,E2 -19139.691} C_VEL
LIN {X 0,Y 256.22,Z 299.163,A -85,B 0,C 180,E1 -19140.53,E2 -19140.53} C_VEL
LIN {X 0,Y 254.264,Z 312.774,A -85,B 0,C 180,E1 -19141.751,E2 -19141.751} C_VEL
LIN {X 0,Y 252.354,Z 324.924,A -85,B 0,C 180,E1 -19143.174,E2 -19143.174} C_VEL
LIN {X 0,Y 250.077,Z 336.489,A -85,B 0,C 180,E1 -19144.848,E2 -19144.848} C_VEL
LIN {X 0,Y 248.331,Z 345.531,A -85,B 0,C 180,E1 -19146.44,E2 -19146.44} C_VEL
LIN {X 0,Y 246.099,Z 355.919,A -85,B 0,C 180,E1 -19148.65,E2 -19148.65} C_VEL
LIN {X 0,Y 244.164,Z 365.303,A -85,B 0,C 180,E1 -19151.109,E2 -19151.109} C_VEL
LIN {X 0,Y 242.708,Z 373.11,A -85,B 0,C 180,E1 -19153.603,E2 -19153.603} C_VEL
LIN {X 0,Y 241.32,Z 380.521,A -85,B 0,C 180,E1 -19156.53,E2 -19156.53} C_VEL
LIN {X 0,Y 240.487,Z 385.695,A -85,B 0,C 180,E1 -19159.052,E2 -19159.052} C_VEL
LIN {X 0,Y 240.071,Z 389.83,A -85,B 0,C 180,E1 -19161.586,E2 -19161.586} C_VEL
LIN {X 0,Y 239.813,Z 393.986,A -85,B 0,C 180,E1 -19164.959,E2 -19164.959} C_VEL
LIN {X 0,Y 239.848,Z 396.667,A -85,B 0,C 180,E1 -19168.323,E2 -19168.323} C_VEL
LIN {X 0,Y 239.921,Z 397.48,A -85,B 0,C 180,E1 -19170.002,E2 -19170.002} C_VEL
LIN {X 0,Y 239.756,Z 398.074,A -85,B 0,C 180,E1 -19173.363,E2 -19173.363} C_VEL
LIN {X 0,Y 239.907,Z 397.344,A -85,B 0,C 180,E1 -19176.732,E2 -19176.732} C_VEL
LIN {X 0,Y 240.5,Z 395.293,A -85,B 0,C 180,E1 -19180.1,E2 -19180.1} C_VEL
LIN {X 0,Y 241.634,Z 391.883,A -85,B 0,C 180,E1 -19183.457,E2 -19183.457} C_VEL
LIN {X 0,Y 243.626,Z 387.018,A -85,B 0,C 180,E1 -19186.769,E2 -19186.769} C_VEL
LIN {X 0,Y 246.242,Z 380.562,A -85,B 0,C 180,E1 -19190.031,E2 -19190.031} C_VEL
LIN {X 0,Y 249.218,Z 373.422,A -85,B 0,C 180,E1 -19192.817,E2 -19192.817} C_VEL
LIN {X 0,Y 252.253,Z 365.98,A -85,B 0,C 180,E1 -19195.145,E2 -19195.145} C_VEL
LIN {X 0,Y 255.732,Z 357.08,A -85,B 0,C 180,E1 -19197.41,E2 -19197.41} C_VEL
LIN {X 0,Y 259.513,Z 346.703,A -85,B 0,C 180,E1 -19199.538,E2 -19199.538} C_VEL
LIN {X 0,Y 262.968,Z 335.961,A -85,B 0,C 180,E1 -19201.322,E2 -19201.322} C_VEL
LIN {X 0,Y 266.221,Z 325.047,A -85,B 0,C 180,E1 -19202.766,E2 -19202.766} C_VEL
LIN {X 0,Y 269.344,Z 312.324,A -85,B 0,C 180,E1 -19204.127,E2 -19204.127} C_VEL
LIN {X 0,Y 272.169,Z 299.104,A -85,B 0,C 180,E1 -19205.183,E2 -19205.183} C_VEL
LIN {X 0,Y 274.489,Z 284.724,A -85,B 0,C 180,E1 -19206.024,E2 -19206.024} C_VEL
LIN {X 0,Y 276.048,Z 270.218,A -85,B 0,C 180,E1 -19206.582,E2 -19206.582} C_VEL
LIN {X 0,Y 279.929,Z 196.639,A -85,B 0,C 180,E1 -19208.463,E2 -19208.463} C_VEL
LIN {X 0,Y 279.356,Z 193.961,A -85,B 0,C 180,E1 -19208.672,E2 -19208.672} C_VEL
LIN {X 0,Y 273.033,Z 179.941,A -85,B 0,C 180,E1 -19210.515,E2 -19210.515} C_VEL
LIN {X 0,Y 266.969,Z 168.268,A -85,B 0,C 180,E1 -19212.358,E2 -19212.358} C_VEL
LIN {X 0,Y 261.544,Z 158.897,A -85,B 0,C 180,E1 -19214.108,E2 -19214.108} C_VEL
LIN {X 0,Y 255.745,Z 149.538,A -85,B 0,C 180,E1 -19216.116,E2 -19216.116} C_VEL
LIN {X 0,Y 251.773,Z 143.621,A -85,B 0,C 180,E1 -19217.585,E2 -19217.585} C_VEL
LIN {X 0,Y 248.047,Z 138.162,A -85,B 0,C 180,E1 -19219.053,E2 -19219.053} C_VEL
LIN {X 0,Y 244.753,Z 133.705,A -85,B 0,C 180,E1 -19220.418,E2 -19220.418} C_VEL
LIN {X 0,Y 244.227,Z 132.596,A -85,B 0,C 180,E1 -19220.717,E2 -19220.717} C_VEL
LIN {X 0,Y 242.013,Z 125.956,A -85,B 0,C 180,E1 -19225.378,E2 -19225.378} C_VEL
LIN {X 0,Y 241.969,Z 125.961,A -85,B 0,C 180,E1 -19228.474,E2 -19228.474} C_VEL
LIN {X 0,Y 241.984,Z 125.957,A -85,B 0,C 180,E1 -19232.305,E2 -19232.305} C_VEL
